LIN {X 0,Y 309.133,Z 1073.835,A -85,B 0,C 180,E1 8987.484,E2 8987.484} C_VEL
LIN {X 0,Y 294.243,Z 1088.868,A -85,B 0,C 180,E1 8985.569,E2 8985.569} C_VEL
LIN {X 0,Y 276.19,Z 1105.751,A -85,B 0,C 180,E1 8982.887,E2 8982.887} C_VEL
LIN {X 0,Y 257.038,Z 1121.964,A -85,B 0,C 180,E1 8979.506,E2 8979.506} C_VEL
LIN {X 0,Y 241.491,Z 1134.247,A -85,B 0,C 180,E1 8976.208,E2 8976.208} C_VEL
LIN {X 0,Y 226.678,Z 1145.297,A -85,B 0,C 180,E1 8972.448,E2 8972.448} C_VEL
LIN {X 0,Y 209.69,Z 1157.432,A -85,B 0,C 180,E1 8967.057,E2 8967.057} C_VEL
LIN {X 0,Y 194.519,Z 1167.62,A -85,B 0,C 180,E1 8960.783,E2 8960.783} C_VEL
LIN {X 0,Y 183.451,Z 1175.062,A -85,B 0,C 180,E1 8954.675,E2 8954.675} C_VEL
LIN {X 0,Y 174.687,Z 1181.102,A -85,B 0,C 180,E1 8948.182,E2 8948.182} C_VEL
LIN {X 0,Y 167.743,Z 1186.26,A -85,B 0,C 180,E1 8940.838,E2 8940.838} C_VEL
LIN {X 0,Y 162.399,Z 1191.034,A -85,B 0,C 180,E1 8931.3,E2 8931.3} C_VEL
LIN {X 0,Y 160.352,Z 1193.692,A -85,B 0,C 180,E1 8922.606,E2 8922.606} C_VEL
LIN {X 0,Y 160.035,Z 1194.885,A -85,B 0,C 180,E1 8915.737,E2 8915.737} C_VEL
LIN {X 0,Y 160.057,Z 1195.249,A -85,B 0,C 180,E1 8909.642,E2 8909.642} C_VEL
LIN {X 0,Y 160.043,Z 1194.803,A -85,B 0,C 180,E1 8903.183,E2 8903.183} C_VEL
LIN {X 0,Y 160.656,Z 1193.192,A -85,B 0,C 180,E1 8895.217,E2 8895.217} C_VEL
LIN {X 0,Y 163.453,Z 1189.886,A -85,B 0,C 180,E1 8886.189,E2 8886.189} C_VEL
LIN {X 0,Y 168.275,Z 1185.792,A -85,B 0,C 180,E1 8878.475,E2 8878.475} C_VEL
LIN {X 0,Y 175.061,Z 1180.789,A -85,B 0,C 180,E1 8871.49,E2 8871.49} C_VEL
LIN {X 0,Y 184.092,Z 1174.573,A -85,B 0,C 180,E1 8864.918,E2 8864.918} C_VEL
LIN {X 0,Y 197.499,Z 1165.629,A -85,B 0,C 180,E1 8857.837,E2 8857.837} C_VEL
LIN {X 0,Y 213.58,Z 1154.53,A -85,B 0,C 180,E1 8851.568,E2 8851.568} C_VEL
LIN {X 0,Y 227.388,Z 1144.675,A -85,B 0,C 180,E1 8847.349,E2 8847.349} C_VEL
LIN {X 0,Y 241.484,Z 1134.135,A -85,B 0,C 180,E1 8843.788,E2 8843.788} C_VEL
LIN {X 0,Y 257.187,Z 1121.707,A -85,B 0,C 180,E1 8840.458,E2 8840.458} C_VEL
LIN {X 0,Y 277.026,Z 1104.8,A -85,B 0,C 180,E1 8836.971,E2 8836.971} C_VEL
LIN {X 0,Y 294.234,Z 1088.677,A -85,B 0,C 180,E1 8834.425,E2 8834.425} C_VEL
LIN {X 0,Y 309.275,Z 1073.464,A -85,B 0,C 180,E1 8832.49,E2 8832.49} C_VEL
LIN {X 0,Y 324.192,Z 1057.141,A -85,B 0,C 180,E1 8830.796,E2 8830.796} C_VEL
LIN {X 0,Y 341.69,Z 1036.137,A -85,B 0,C 180,E1 8829.035,E2 8829.035} C_VEL
LIN {X 0,Y 356.653,Z 1015.961,A -85,B 0,C 180,E1 8827.687,E2 8827.687} C_VEL
LIN {X 0,Y 368.714,Z 998.106,A -85,B 0,C 180,E1 8826.696,E2 8826.696} C_VEL
LIN {X 0,Y 379.924,Z 979.871,A -85,B 0,C 180,E1 8825.85,E2 8825.85} C_VEL
LIN {X 0,Y 390.494,Z 960.848,A -85,B 0,C 180,E1 8825.108,E2 8825.108} C_VEL
LIN {X 0,Y 401.796,Z 938.038,A -85,B 0,C 180,E1 8824.371,E2 8824.371} C_VEL
LIN {X 0,Y 412.803,Z 911.976,A -85,B 0,C 180,E1 8823.706,E2 8823.706} C_VEL
LIN {X 0,Y 420.62,Z 890.255,A -85,B 0,C 180,E1 8823.261,E2 8823.261} C_VEL
LIN {X 0,Y 427.238,Z 868.633,A -85,B 0,C 180,E1 8822.905,E2 8822.905} C_VEL
LIN {X 0,Y 433.159,Z 845.153,A -85,B 0,C 180,E1 8822.584,E2 8822.584} C_VEL
LIN {X 0,Y 438.789,Z 815.012,A -85,B 0,C 180,E1 8822.194,E2 8822.194} C_VEL
LIN {X 0,Y 446.722,Z 751.327,A -85,B 0,C 180,E1 8821.414,E2 8821.414} C_VEL
LIN {X 0,Y 455.842,Z 675.807,A -85,B 0,C 180,E1 8820.471,E2 8820.471} C_VEL
LIN {X 0,Y 455.856,Z 675.472,A -85,B 0,C 180,E1 8819.372,E2 8819.372} C_VEL
LIN {X 0,Y 455.813,Z 675.985,A -85,B 0,C 180,E1 8819.103,E2 8819.103} C_VEL
LIN {X 0,Y 439.212,Z 811.582,A -85,B 0,C 180,E1 8817.459,E2 8817.459} C_VEL
LIN {X 0,Y 434.453,Z 838.722,A -85,B 0,C 180,E1 8817.116,E2 8817.116} C_VEL
LIN {X 0,Y 427.865,Z 865.427,A -85,B 0,C 180,E1 8816.703,E2 8816.703} C_VEL
LIN {X 0,Y 421.567,Z 886.299,A -85,B 0,C 180,E1 8816.301,E2 8816.301} C_VEL
LIN {X 0,Y 414.352,Z 906.676,A -85,B 0,C 180,E1 8815.831,E2 8815.831} C_VEL
LIN {X 0,Y 405.832,Z 927.534,A -85,B 0,C 180,E1 8815.256,E2 8815.256} C_VEL
LIN {X 0,Y 394.302,Z 952.101,A -85,B 0,C 180,E1 8814.434,E2 8814.434} C_VEL
LIN {X 0,Y 381.896,Z 974.697,A -85,B 0,C 180,E1 8813.505,E2 8813.505} C_VEL
LIN {X 0,Y 370.033,Z 994.026,A -85,B 0,C 180,E1 8812.547,E2 8812.547} C_VEL
LIN {X 0,Y 358.475,Z 1011.099,A -85,B 0,C 180,E1 8811.55,E2 8811.55} C_VEL
LIN {X 0,Y 344.895,Z 1029.371,A -85,B 0,C 180,E1 8810.287,E2 8810.287} C_VEL
LIN {X 0,Y 326.629,Z 1051.422,A -85,B 0,C 180,E1 8808.397,E2 8808.397} C_VEL
LIN {X 0,Y 311.406,Z 1067.929,A -85,B 0,C 180,E1 8806.622,E2 8806.622} C_VEL
LIN {X 0,Y 297.374,Z 1081.972,A -85,B 0,C 180,E1 8804.791,E2 8804.791} C_VEL
LIN {X 0,Y 282.808,Z 1095.479,A -85,B 0,C 180,E1 8802.663,E2 8802.663} C_VEL
LIN {X 0,Y 267.028,Z 1109.062,A -85,B 0,C 180,E1 8800.025,E2 8800.025} C_VEL
LIN {X 0,Y 247.214,Z 1124.737,A -85,B 0,C 180,E1 8796.072,E2 8796.072} C_VEL
LIN {X 0,Y 231.552,Z 1136.124,A -85,B 0,C 180,E1 8792.276,E2 8792.276} C_VEL
LIN {X 0,Y 217.635,Z 1145.68,A -85,B 0,C 180,E1 8788.203,E2 8788.203} C_VEL
LIN {X 0,Y 204.25,Z 1154.443,A -85,B 0,C 180,E1 8783.4,E2 8783.4} C_VEL
LIN {X 0,Y 189.786,Z 1163.686,A -85,B 0,C 180,E1 8776.638,E2 8776.638} C_VEL
LIN {X 0,Y 177.958,Z 1170.967,A -85,B 0,C 180,E1 8768.996,E2 8768.996} C_VEL
LIN {X 0,Y 170.605,Z 1175.705,A -85,B 0,C 180,E1 8762.23,E2 8762.23} C_VEL
LIN {X 0,Y 165.299,Z 1179.405,A -85,B 0,C 180,E1 8755.05,E2 8755.05} C_VEL
LIN {X 0,Y 162.12,Z 1181.995,A -85,B 0,C 180,E1 8747.961,E2 8747.961} C_VEL
LIN {X 0,Y 160.603,Z 1183.636,A -85,B 0,C 180,E1 8741.128,E2 8741.128} C_VEL
LIN {X 0,Y 160.127,Z 1184.462,A -85,B 0,C 180,E1 8735.015,E2 8735.015} C_VEL
LIN {X 0,Y 160.068,Z 1184.682,A -85,B 0,C 180,E1 8728.568,E2 8728.568} C_VEL
LIN {X 0,Y 160.302,Z 1184.173,A -85,B 0,C 180,E1 8721.752,E2 8721.752} C_VEL
LIN {X 0,Y 161.666,Z 1182.47,A -85,B 0,C 180,E1 8713.469,E2 8713.469} C_VEL
LIN {X 0,Y 164.853,Z 1179.775,A -85,B 0,C 180,E1 8705.643,E2 8705.643} C_VEL
LIN {X 0,Y 169.941,Z 1176.184,A -85,B 0,C 180,E1 8698.424,E2 8698.424} C_VEL
LIN {X 0,Y 177.089,Z 1171.558,A -85,B 0,C 180,E1 8691.606,E2 8691.606} C_VEL
LIN {X 0,Y 186.7,Z 1165.567,A -85,B 0,C 180,E1 8685.016,E2 8685.016} C_VEL
LIN {X 0,Y 200.602,Z 1156.965,A -85,B 0,C 180,E1 8678.046,E2 8678.046} C_VEL
LIN {X 0,Y 216.185,Z 1146.747,A -85,B 0,C 180,E1 8672.181,E2 8672.181} C_VEL
LIN {X 0,Y 230.378,Z 1137.051,A -85,B 0,C 180,E1 8667.953,E2 8667.953} C_VEL
LIN {X 0,Y 245.568,Z 1126.068,A -85,B 0,C 180,E1 8664.211,E2 8664.211} C_VEL
LIN {X 0,Y 264.596,Z 1111.293,A -85,B 0,C 180,E1 8660.345,E2 8660.345} C_VEL
LIN {X 0,Y 281.866,Z 1096.514,A -85,B 0,C 180,E1 8657.405,E2 8657.405} C_VEL
LIN {X 0,Y 296.484,Z 1083.035,A -85,B 0,C 180,E1 8655.251,E2 8655.251} C_VEL
LIN {X 0,Y 311.317,Z 1068.251,A -85,B 0,C 180,E1 8653.309,E2 8653.309} C_VEL
LIN {X 0,Y 327.453,Z 1050.768,A -85,B 0,C 180,E1 8651.435,E2 8651.435} C_VEL
LIN {X 0,Y 345.095,Z 1029.428,A -85,B 0,C 180,E1 8649.615,E2 8649.615} C_VEL
LIN {X 0,Y 358.749,Z 1011.07,A -85,B 0,C 180,E1 8648.347,E2 8648.347} C_VEL
LIN {X 0,Y 370.481,Z 993.735,A -85,B 0,C 180,E1 8647.338,E2 8647.338} C_VEL
LIN {X 0,Y 382.316,Z 974.425,A -85,B 0,C 180,E1 8646.385,E2 8646.385} C_VEL
LIN {X 0,Y 395.69,Z 949.815,A -85,B 0,C 180,E1 8645.387,E2 8645.387} C_VEL
LIN {X 0,Y 406.271,Z 927.122,A -85,B 0,C 180,E1 8644.638,E2 8644.638} C_VEL
LIN {X 0,Y 414.492,Z 907.01,A -85,B 0,C 180,E1 8644.083,E2 8644.083} C_VEL
LIN {X 0,Y 421.775,Z 886.483,A -85,B 0,C 180,E1 8643.61,E2 8643.61} C_VEL
LIN {X 0,Y 428.306,Z 864.819,A -85,B 0,C 180,E1 8643.194,E2 8643.194} C_VEL
LIN {X 0,Y 434.947,Z 837.545,A -85,B 0,C 180,E1 8642.777,E2 8642.777} C_VEL
LIN {X 0,Y 439.509,Z 811.419,A -85,B 0,C 180,E1 8642.447,E2 8642.447} C_VEL
LIN {X 0,Y 456.081,Z 676.099,A -85,B 0,C 180,E1 8640.786,E2 8640.786} C_VEL
LIN {X 0,Y 456.119,Z 675.624,A -85,B 0,C 180,E1 8640,E2 8640} C_VEL
LIN {X 0,Y 456.064,Z 676.332,A -85,B 0,C 180,E1 8639.494,E2 8639.494} C_VEL
LIN {X 0,Y 447.534,Z 746.879,A -85,B 0,C 180,E1 8638.641,E2 8638.641} C_VEL
LIN {X 0,Y 446.581,Z 754.582,A -85,B 0,C 180,E1 8638.675,E2 8638.675} C_VEL
LIN {X 0,Y 443.952,Z 775.216,A -85,B 0,C 180,E1 8639.235,E2 8639.235} C_VEL
LIN {X 0,Y 443.138,Z 781.824,A -85,B 0,C 180,E1 8639.253,E2 8639.253} C_VEL
LIN {X 0,Y 437.817,Z 821.436,A -85,B 0,C 180,E1 8638.777,E2 8638.777} C_VEL
LIN {X 0,Y 432.44,Z 847.855,A -85,B 0,C 180,E1 8638.445,E2 8638.445} C_VEL
LIN {X 0,Y 426.753,Z 869.852,A -85,B 0,C 180,E1 8638.156,E2 8638.156} C_VEL
LIN {X 0,Y 420.056,Z 891.346,A -85,B 0,C 180,E1 8637.817,E2 8637.817} C_VEL
LIN {X 0,Y 410.398,Z 917.489,A -85,B 0,C 180,E1 8637.295,E2 8637.295} C_VEL
LIN {X 0,Y 399.613,Z 941.699,A -85,B 0,C 180,E1 8636.679,E2 8636.679} C_VEL
LIN {X 0,Y 389.37,Z 961.953,A -85,B 0,C 180,E1 8636.044,E2 8636.044} C_VEL
LIN {X 0,Y 378.147,Z 981.776,A -85,B 0,C 180,E1 8635.298,E2 8635.298} C_VEL
LIN {X 0,Y 364.255,Z 1003.777,A -85,B 0,C 180,E1 8634.289,E2 8634.289} C_VEL
LIN {X 0,Y 347.814,Z 1026.636,A -85,B 0,C 180,E1 8632.978,E2 8632.978} C_VEL
LIN {X 0,Y 333.928,Z 1044.093,A -85,B 0,C 180,E1 8631.736,E2 8631.736} C_VEL
LIN {X 0,Y 320.189,Z 1059.945,A -85,B 0,C 180,E1 8630.383,E2 8630.383} C_VEL
LIN {X 0,Y 304.863,Z 1076.22,A -85,B 0,C 180,E1 8628.704,E2 8628.704} C_VEL
LIN {X 0,Y 285.175,Z 1095.312,A -85,B 0,C 180,E1 8626.206,E2 8626.206} C_VEL
LIN {X 0,Y 267.821,Z 1110.53,A -85,B 0,C 180,E1 8623.629,E2 8623.629} C_VEL
LIN {X 0,Y 251.898,Z 1123.505,A -85,B 0,C 180,E1 8620.855,E2 8620.855} C_VEL
LIN {X 0,Y 235.856,Z 1135.727,A -85,B 0,C 180,E1 8617.542,E2 8617.542} C_VEL
LIN {X 0,Y 217.054,Z 1149.161,A -85,B 0,C 180,E1 8612.754,E2 8612.754} C_VEL
LIN {X 0,Y 200.577,Z 1160.078,A -85,B 0,C 180,E1 8607.399,E2 8607.399} C_VEL
LIN {X 0,Y 187.713,Z 1168.338,A -85,B 0,C 180,E1 8602.029,E2 8602.029} C_VEL
LIN {X 0,Y 176.096,Z 1175.728,A -85,B 0,C 180,E1 8595.677,E2 8595.677} C_VEL
LIN {X 0,Y 164.807,Z 1183.173,A -85,B 0,C 180,E1 8586.914,E2 8586.914} C_VEL
LIN {X 0,Y 157.356,Z 1188.463,A -85,B 0,C 180,E1 8577.636,E2 8577.636} C_VEL
LIN {X 0,Y 153.824,Z 1191.615,A -85,B 0,C 180,E1 8569.755,E2 8569.755} C_VEL
LIN {X 0,Y 152.3,Z 1193.647,A -85,B 0,C 180,E1 8562.127,E2 8562.127} C_VEL
LIN {X 0,Y 152.038,Z 1194.648,A -85,B 0,C 180,E1 8555.661,E2 8555.661} C_VEL
LIN {X 0,Y 152.06,Z 1194.963,A -85,B 0,C 180,E1 8549.246,E2 8549.246} C_VEL
LIN {X 0,Y 152.062,Z 1194.506,A -85,B 0,C 180,E1 8542.443,E2 8542.443} C_VEL
LIN {X 0,Y 152.934,Z 1192.683,A -85,B 0,C 180,E1 8533.673,E2 8533.673} C_VEL
LIN {X 0,Y 155.921,Z 1189.614,A -85,B 0,C 180,E1 8524.961,E2 8524.961} C_VEL
LIN {X 0,Y 161.222,Z 1185.518,A -85,B 0,C 180,E1 8516.924,E2 8516.924} C_VEL
LIN {X 0,Y 168.569,Z 1180.517,A -85,B 0,C 180,E1 8509.72,E2 8509.72} C_VEL
LIN {X 0,Y 178.049,Z 1174.414,A -85,B 0,C 180,E1 8503.111,E2 8503.111} C_VEL
LIN {X 0,Y 191.23,Z 1166.08,A -85,B 0,C 180,E1 8496.371,E2 8496.371} C_VEL
LIN {X 0,Y 208.586,Z 1154.721,A -85,B 0,C 180,E1 8489.817,E2 8489.817} C_VEL
LIN {X 0,Y 223.687,Z 1144.357,A -85,B 0,C 180,E1 8485.412,E2 8485.412} C_VEL
LIN {X 0,Y 238.203,Z 1133.856,A -85,B 0,C 180,E1 8481.929,E2 8481.929} C_VEL
LIN {X 0,Y 254.364,Z 1121.429,A -85,B 0,C 180,E1 8478.68,E2 8478.68} C_VEL
LIN {X 0,Y 274.693,Z 1104.522,A -85,B 0,C 180,E1 8475.297,E2 8475.297} C_VEL
LIN {X 0,Y 292.263,Z 1088.4,A -85,B 0,C 180,E1 8472.836,E2 8472.836} C_VEL
LIN {X 0,Y 307.578,Z 1073.188,A -85,B 0,C 180,E1 8470.972,E2 8470.972} C_VEL
LIN {X 0,Y 322.534,Z 1057.09,A -85,B 0,C 180,E1 8469.365,E2 8469.365} C_VEL
LIN {X 0,Y 340.019,Z 1036.476,A -85,B 0,C 180,E1 8467.702,E2 8467.702} C_VEL
LIN {X 0,Y 355.458,Z 1015.952,A -85,B 0,C 180,E1 8466.387,E2 8466.387} C_VEL
LIN {X 0,Y 368.085,Z 997.464,A -85,B 0,C 180,E1 8465.409,E2 8465.409} C_VEL
LIN {X 0,Y 379.661,Z 978.78,A -85,B 0,C 180,E1 8464.587,E2 8464.587} C_VEL
LIN {X 0,Y 391.362,Z 957.767,A -85,B 0,C 180,E1 8463.819,E2 8463.819} C_VEL
LIN {X 0,Y 404.015,Z 931.651,A -85,B 0,C 180,E1 8463.053,E2 8463.053} C_VEL
LIN {X 0,Y 413.342,Z 909.121,A -85,B 0,C 180,E1 8462.528,E2 8462.528} C_VEL
LIN {X 0,Y 420.591,Z 888.917,A -85,B 0,C 180,E1 8462.143,E2 8462.143} C_VEL
LIN {X 0,Y 427.152,Z 867.489,A -85,B 0,C 180,E1 8461.813,E2 8461.813} C_VEL
LIN {X 0,Y 433.674,Z 841.477,A -85,B 0,C 180,E1 8461.475,E2 8461.475} C_VEL
LIN {X 0,Y 438.74,Z 813.437,A -85,B 0,C 180,E1 8461.126,E2 8461.126} C_VEL
LIN {X 0,Y 449.767,Z 725.044,A -85,B 0,C 180,E1 8460.073,E2 8460.073} C_VEL
LIN {X 0,Y 452.539,Z 702.413,A -85,B 0,C 180,E1 8459.801,E2 8459.801} C_VEL
LIN {X 0,Y 438.884,Z 812.187,A -85,B 0,C 180,E1 8458.499,E2 8458.499} C_VEL
LIN {X 0,Y 433.988,Z 839.631,A -85,B 0,C 180,E1 8458.163,E2 8458.163} C_VEL
LIN {X 0,Y 427.417,Z 865.917,A -85,B 0,C 180,E1 8457.773,E2 8457.773} C_VEL
LIN {X 0,Y 421.125,Z 886.572,A -85,B 0,C 180,E1 8457.392,E2 8457.392} C_VEL
LIN {X 0,Y 413.79,Z 907.091,A -85,B 0,C 180,E1 8456.939,E2 8456.939} C_VEL
LIN {X 0,Y 405.245,Z 927.806,A -85,B 0,C 180,E1 8456.392,E2 8456.392} C_VEL
LIN {X 0,Y 393.601,Z 952.371,A -85,B 0,C 180,E1 8455.605,E2 8455.605} C_VEL
LIN {X 0,Y 380.583,Z 975.773,A -85,B 0,C 180,E1 8454.682,E2 8454.682} C_VEL
LIN {X 0,Y 369.104,Z 994.24,A -85,B 0,C 180,E1 8453.802,E2 8453.802} C_VEL
LIN {X 0,Y 357.239,Z 1011.55,A -85,B 0,C 180,E1 8452.834,E2 8452.834} C_VEL
LIN {X 0,Y 343.142,Z 1030.245,A -85,B 0,C 180,E1 8451.588,E2 8451.588} C_VEL
LIN {X 0,Y 324.158,Z 1052.696,A -85,B 0,C 180,E1 8449.719,E2 8449.719} C_VEL
LIN {X 0,Y 309.168,Z 1068.643,A -85,B 0,C 180,E1 8448.054,E2 8448.054} C_VEL
LIN {X 0,Y 294.43,Z 1083.078,A -85,B 0,C 180,E1 8446.223,E2 8446.223} C_VEL
LIN {X 0,Y 278.729,Z 1097.27,A -85,B 0,C 180,E1 8444.022,E2 8444.022} C_VEL
LIN {X 0,Y 259.332,Z 1113.38,A -85,B 0,C 180,E1 8440.839,E2 8440.839} C_VEL
LIN {X 0,Y 241.587,Z 1126.697,A -85,B 0,C 180,E1 8437.358,E2 8437.358} C_VEL
LIN {X 0,Y 226.303,Z 1137.406,A -85,B 0,C 180,E1 8433.753,E2 8433.753} C_VEL
LIN {X 0,Y 211.971,Z 1146.85,A -85,B 0,C 180,E1 8429.678,E2 8429.678} C_VEL
LIN {X 0,Y 195.666,Z 1157.081,A -85,B 0,C 180,E1 8423.841,E2 8423.841} C_VEL
LIN {X 0,Y 180.793,Z 1165.837,A -85,B 0,C 180,E1 8416.702,E2 8416.702} C_VEL
LIN {X 0,Y 170.741,Z 1171.729,A -85,B 0,C 180,E1 8410.103,E2 8410.103} C_VEL
LIN {X 0,Y 163.029,Z 1176.372,A -85,B 0,C 180,E1 8403.082,E2 8403.082} C_VEL
LIN {X 0,Y 157.245,Z 1180.13,A -85,B 0,C 180,E1 8395.216,E2 8395.216} C_VEL
LIN {X 0,Y 153.683,Z 1182.906,A -85,B 0,C 180,E1 8386.634,E2 8386.634} C_VEL
LIN {X 0,Y 152.289,Z 1184.538,A -85,B 0,C 180,E1 8377.925,E2 8377.925} C_VEL
LIN {X 0,Y 152.068,Z 1184.979,A -85,B 0,C 180,E1 8370.753,E2 8370.753} C_VEL
LIN {X 0,Y 152.168,Z 1184.695,A -85,B 0,C 180,E1 8363.965,E2 8363.965} C_VEL
LIN {X 0,Y 153.046,Z 1183.553,A -85,B 0,C 180,E1 8356.012,E2 8356.012} C_VEL
LIN {X 0,Y 156.409,Z 1180.803,A -85,B 0,C 180,E1 8346.251,E2 8346.251} C_VEL
LIN {X 0,Y 162.424,Z 1176.793,A -85,B 0,C 180,E1 8337.499,E2 8337.499} C_VEL
LIN {X 0,Y 170.245,Z 1172.074,A -85,B 0,C 180,E1 8330.196,E2 8330.196} C_VEL
LIN {X 0,Y 179.885,Z 1166.425,A -85,B 0,C 180,E1 8323.732,E2 8323.732} C_VEL
LIN {X 0,Y 192.557,Z 1158.974,A -85,B 0,C 180,E1 8317.396,E2 8317.396} C_VEL
LIN {X 0,Y 210.484,Z 1147.915,A -85,B 0,C 180,E1 8310.706,E2 8310.706} C_VEL
LIN {X 0,Y 225.875,Z 1137.807,A -85,B 0,C 180,E1 8306.275,E2 8306.275} C_VEL
LIN {X 0,Y 240.913,Z 1127.307,A -85,B 0,C 180,E1 8302.705,E2 8302.705} C_VEL
LIN {X 0,Y 257.581,Z 1114.852,A -85,B 0,C 180,E1 8299.395,E2 8299.395} C_VEL
LIN {X 0,Y 277.778,Z 1098.3,A -85,B 0,C 180,E1 8296.042,E2 8296.042} C_VEL
LIN {X 0,Y 293.784,Z 1083.901,A -85,B 0,C 180,E1 8293.783,E2 8293.783} C_VEL
LIN {X 0,Y 308.622,Z 1069.432,A -85,B 0,C 180,E1 8291.93,E2 8291.93} C_VEL
LIN {X 0,Y 323.765,Z 1053.386,A -85,B 0,C 180,E1 8290.243,E2 8290.243} C_VEL
LIN {X 0,Y 341.679,Z 1032.458,A -85,B 0,C 180,E1 8288.472,E2 8288.472} C_VEL
LIN {X 0,Y 356.71,Z 1012.656,A -85,B 0,C 180,E1 8287.135,E2 8287.135} C_VEL
LIN {X 0,Y 368.576,Z 995.454,A -85,B 0,C 180,E1 8286.162,E2 8286.162} C_VEL
LIN {X 0,Y 380.009,Z 977.185,A -85,B 0,C 180,E1 8285.284,E2 8285.284} C_VEL
LIN {X 0,Y 390.773,Z 958.083,A -85,B 0,C 180,E1 8284.508,E2 8284.508} C_VEL
LIN {X 0,Y 402.781,Z 934.091,A -85,B 0,C 180,E1 8283.699,E2 8283.699} C_VEL
LIN {X 0,Y 413.183,Z 909.393,A -85,B 0,C 180,E1 8283.024,E2 8283.024} C_VEL
LIN {X 0,Y 420.855,Z 888.21,A -85,B 0,C 180,E1 8282.549,E2 8282.549} C_VEL
LIN {X 0,Y 427.316,Z 867.242,A -85,B 0,C 180,E1 8282.158,E2 8282.158} C_VEL
LIN {X 0,Y 433.051,Z 844.755,A -85,B 0,C 180,E1 8281.815,E2 8281.815} C_VEL
LIN {X 0,Y 438.774,Z 814.893,A -85,B 0,C 180,E1 8281.442,E2 8281.442} C_VEL
LIN {X 0,Y 445.925,Z 758.797,A -85,B 0,C 180,E1 8280.774,E2 8280.774} C_VEL
LIN {X 0,Y 452.345,Z 706.338,A -85,B 0,C 180,E1 8280.15,E2 8280.15} C_VEL
LIN {X 0,Y 443.138,Z 781.824,A -85,B 0,C 180,E1 8279.253,E2 8279.253} C_VEL
LIN {X 0,Y 442.206,Z 789.524,A -85,B 0,C 180,E1 8279.294,E2 8279.294} C_VEL
LIN {X 0,Y 439.396,Z 810.123,A -85,B 0,C 180,E1 8279.867,E2 8279.867} C_VEL
LIN {X 0,Y 438.423,Z 816.713,A -85,B 0,C 180,E1 8279.884,E2 8279.884} C_VEL
LIN {X 0,Y 432.733,Z 845.774,A -85,B 0,C 180,E1 8279.534,E2 8279.534} C_VEL
LIN {X 0,Y 426.874,Z 868.532,A -85,B 0,C 180,E1 8279.252,E2 8279.252} C_VEL
LIN {X 0,Y 420.383,Z 889.422,A -85,B 0,C 180,E1 8278.946,E2 8278.946} C_VEL
LIN {X 0,Y 412.571,Z 910.848,A -85,B 0,C 180,E1 8278.556,E2 8278.556} C_VEL
LIN {X 0,Y 401.198,Z 937.398,A -85,B 0,C 180,E1 8277.951,E2 8277.951} C_VEL
LIN {X 0,Y 389.875,Z 959.878,A -85,B 0,C 180,E1 8277.302,E2 8277.302} C_VEL
LIN {X 0,Y 379.099,Z 978.945,A -85,B 0,C 180,E1 8276.634,E2 8276.634} C_VEL
LIN {X 0,Y 367.388,Z 997.617,A -85,B 0,C 180,E1 8275.854,E2 8275.854} C_VEL
LIN {X 0,Y 353.868,Z 1017.113,A -85,B 0,C 180,E1 8274.866,E2 8274.866} C_VEL
LIN {X 0,Y 336.157,Z 1039.909,A -85,B 0,C 180,E1 8273.432,E2 8273.432} C_VEL
LIN {X 0,Y 320.61,Z 1057.808,A -85,B 0,C 180,E1 8272.024,E2 8272.024} C_VEL
LIN {X 0,Y 305.578,Z 1073.672,A -85,B 0,C 180,E1 8270.496,E2 8270.496} C_VEL
LIN {X 0,Y 289.583,Z 1089.215,A -85,B 0,C 180,E1 8268.649,E2 8268.649} C_VEL
LIN {X 0,Y 269.96,Z 1106.694,A -85,B 0,C 180,E1 8266.018,E2 8266.018} C_VEL
LIN {X 0,Y 250.952,Z 1121.936,A -85,B 0,C 180,E1 8262.983,E2 8262.983} C_VEL
LIN {X 0,Y 235.188,Z 1133.696,A -85,B 0,C 180,E1 8259.974,E2 8259.974} C_VEL
LIN {X 0,Y 219.288,Z 1144.804,A -85,B 0,C 180,E1 8256.343,E2 8256.343} C_VEL
LIN {X 0,Y 200.986,Z 1156.879,A -85,B 0,C 180,E1 8251.111,E2 8251.111} C_VEL
LIN {X 0,Y 184.478,Z 1166.968,A -85,B 0,C 180,E1 8244.926,E2 8244.926} C_VEL
LIN {X 0,Y 171.871,Z 1174.51,A -85,B 0,C 180,E1 8238.63,E2 8238.63} C_VEL
LIN {X 0,Y 161.828,Z 1180.552,A -85,B 0,C 180,E1 8231.857,E2 8231.857} C_VEL
LIN {X 0,Y 153.35,Z 1185.93,A -85,B 0,C 180,E1 8223.656,E2 8223.656} C_VEL
LIN {X 0,Y 146.994,Z 1190.615,A -85,B 0,C 180,E1 8213.236,E2 8213.236} C_VEL
LIN {X 0,Y 144.513,Z 1193.158,A -85,B 0,C 180,E1 8204.014,E2 8204.014} C_VEL
LIN {X 0,Y 144.045,Z 1194.358,A -85,B 0,C 180,E1 8196.376,E2 8196.376} C_VEL
LIN {X 0,Y 144.065,Z 1194.724,A -85,B 0,C 180,E1 8189.602,E2 8189.602} C_VEL
LIN {X 0,Y 144.055,Z 1194.301,A -85,B 0,C 180,E1 8182.823,E2 8182.823} C_VEL
LIN {X 0,Y 144.847,Z 1192.768,A -85,B 0,C 180,E1 8173.972,E2 8173.972} C_VEL
LIN {X 0,Y 148.469,Z 1189.342,A -85,B 0,C 180,E1 8163.61,E2 8163.61} C_VEL
LIN {X 0,Y 154.293,Z 1185.243,A -85,B 0,C 180,E1 8155.232,E2 8155.232} C_VEL
LIN {X 0,Y 162.554,Z 1180.06,A -85,B 0,C 180,E1 8147.573,E2 8147.573} C_VEL
LIN {X 0,Y 172.925,Z 1173.822,A -85,B 0,C 180,E1 8140.761,E2 8140.761} C_VEL
LIN {X 0,Y 188.241,Z 1164.705,A -85,B 0,C 180,E1 8133.497,E2 8133.497} C_VEL
LIN {X 0,Y 205.231,Z 1153.972,A -85,B 0,C 180,E1 8127.541,E2 8127.541} C_VEL
LIN {X 0,Y 220.138,Z 1144.117,A -85,B 0,C 180,E1 8123.441,E2 8123.441} C_VEL
LIN {X 0,Y 235.181,Z 1133.578,A -85,B 0,C 180,E1 8120.021,E2 8120.021} C_VEL
LIN {X 0,Y 251.92,Z 1121.054,A -85,B 0,C 180,E1 8116.843,E2 8116.843} C_VEL
LIN {X 0,Y 272.81,Z 1104.059,A -85,B 0,C 180,E1 8113.566,E2 8113.566} C_VEL
LIN {X 0,Y 290.52,Z 1088.123,A -85,B 0,C 180,E1 8111.229,E2 8111.229} C_VEL
LIN {X 0,Y 306.101,Z 1072.911,A -85,B 0,C 180,E1 8109.44,E2 8109.44} C_VEL
LIN {X 0,Y 321.72,Z 1056.338,A -85,B 0,C 180,E1 8107.86,E2 8107.86} C_VEL
LIN {X 0,Y 339.96,Z 1034.971,A -85,B 0,C 180,E1 8106.232,E2 8106.232} C_VEL
LIN {X 0,Y 354.826,Z 1015.412,A -85,B 0,C 180,E1 8105.051,E2 8105.051} C_VEL
LIN {X 0,Y 367.208,Z 997.487,A -85,B 0,C 180,E1 8104.148,E2 8104.148} C_VEL
LIN {X 0,Y 378.606,Z 979.324,A -85,B 0,C 180,E1 8103.386,E2 8103.386} C_VEL
LIN {X 0,Y 389.381,Z 960.301,A -85,B 0,C 180,E1 8102.717,E2 8102.717} C_VEL
LIN {X 0,Y 400.702,Z 937.866,A -85,B 0,C 180,E1 8102.065,E2 8102.065} C_VEL
LIN {X 0,Y 412.074,Z 911.428,A -85,B 0,C 180,E1 8101.458,E2 8101.458} C_VEL
LIN {X 0,Y 420.011,Z 889.706,A -85,B 0,C 180,E1 8101.06,E2 8101.06} C_VEL
LIN {X 0,Y 426.689,Z 868.206,A -85,B 0,C 180,E1 8100.746,E2 8100.746} C_VEL
LIN {X 0,Y 432.67,Z 844.86,A -85,B 0,C 180,E1 8100.456,E2 8100.456} C_VEL
LIN {X 0,Y 438.452,Z 814.548,A -85,B 0,C 180,E1 8100.091,E2 8100.091} C_VEL
LIN {X 0,Y 441.751,Z 790.273,A -85,B 0,C 180,E1 8099.803,E2 8099.803} C_VEL
LIN {X 0,Y 436.617,Z 825.351,A -85,B 0,C 180,E1 8099.394,E2 8099.394} C_VEL
LIN {X 0,Y 431.802,Z 848.29,A -85,B 0,C 180,E1 8099.11,E2 8099.11} C_VEL
LIN {X 0,Y 426.226,Z 869.517,A -85,B 0,C 180,E1 8098.794,E2 8098.794} C_VEL
LIN {X 0,Y 419.353,Z 891.263,A -85,B 0,C 180,E1 8098.398,E2 8098.398} C_VEL
LIN {X 0,Y 409.243,Z 917.962,A -85,B 0,C 180,E1 8097.797,E2 8097.797} C_VEL
LIN {X 0,Y 398.973,Z 940.651,A -85,B 0,C 180,E1 8097.164,E2 8097.164} C_VEL
LIN {X 0,Y 389.157,Z 959.792,A -85,B 0,C 180,E1 8096.529,E2 8096.529} C_VEL
LIN {X 0,Y 378.533,Z 978.342,A -85,B 0,C 180,E1 8095.803,E2 8095.803} C_VEL
LIN {X 0,Y 366.389,Z 997.425,A -85,B 0,C 180,E1 8094.915,E2 8094.915} C_VEL
LIN {X 0,Y 350.704,Z 1019.538,A -85,B 0,C 180,E1 8093.669,E2 8093.669} C_VEL
LIN {X 0,Y 334.555,Z 1039.558,A -85,B 0,C 180,E1 8092.271,E2 8092.271} C_VEL
LIN {X 0,Y 320.003,Z 1055.973,A -85,B 0,C 180,E1 8090.876,E2 8090.876} C_VEL
LIN {X 0,Y 305.265,Z 1071.216,A -85,B 0,C 180,E1 8089.299,E2 8089.299} C_VEL
LIN {X 0,Y 288.089,Z 1087.516,A -85,B 0,C 180,E1 8087.226,E2 8087.226} C_VEL
LIN {X 0,Y 267.84,Z 1104.792,A -85,B 0,C 180,E1 8084.391,E2 8084.391} C_VEL
LIN {X 0,Y 251.56,Z 1117.475,A -85,B 0,C 180,E1 8081.699,E2 8081.699} C_VEL
LIN {X 0,Y 236.087,Z 1128.657,A -85,B 0,C 180,E1 8078.705,E2 8078.705} C_VEL
LIN {X 0,Y 220.01,Z 1139.482,A -85,B 0,C 180,E1 8074.997,E2 8074.997} C_VEL
LIN {X 0,Y 200.845,Z 1151.45,A -85,B 0,C 180,E1 8069.456,E2 8069.456} C_VEL
LIN {X 0,Y 185.401,Z 1160.387,A -85,B 0,C 180,E1 8063.612,E2 8063.612} C_VEL
LIN {X 0,Y 173.261,Z 1167.165,A -85,B 0,C 180,E1 8057.618,E2 8057.618} C_VEL
LIN {X 0,Y 162.727,Z 1172.981,A -85,B 0,C 180,E1 8050.64,E2 8050.64} C_VEL
LIN {X 0,Y 152.993,Z 1178.584,A -85,B 0,C 180,E1 8041.084,E2 8041.084} C_VEL
LIN {X 0,Y 147.146,Z 1182.211,A -85,B 0,C 180,E1 8031.108,E2 8031.108} C_VEL
LIN {X 0,Y 144.901,Z 1184.041,A -85,B 0,C 180,E1 8023.162,E2 8023.162} C_VEL
LIN {X 0,Y 144.155,Z 1184.989,A -85,B 0,C 180,E1 8015.572,E2 8015.572} C_VEL
LIN {X 0,Y 144.073,Z 1185.229,A -85,B 0,C 180,E1 8008.807,E2 8008.807} C_VEL
LIN {X 0,Y 144.346,Z 1184.766,A -85,B 0,C 180,E1 8001.235,E2 8001.235} C_VEL
LIN {X 0,Y 146.007,Z 1183.112,A -85,B 0,C 180,E1 7992.052,E2 7992.052} C_VEL
LIN {X 0,Y 149.822,Z 1180.457,A -85,B 0,C 180,E1 7983.419,E2 7983.419} C_VEL
LIN {X 0,Y 156.106,Z 1176.725,A -85,B 0,C 180,E1 7975.247,E2 7975.247} C_VEL
LIN {X 0,Y 164.704,Z 1171.935,A -85,B 0,C 180,E1 7967.786,E2 7967.786} C_VEL
LIN {X 0,Y 176.413,Z 1165.527,A -85,B 0,C 180,E1 7960.583,E2 7960.583} C_VEL
LIN {X 0,Y 193.349,Z 1155.934,A -85,B 0,C 180,E1 7953.097,E2 7953.097} C_VEL
LIN {X 0,Y 208.499,Z 1146.844,A -85,B 0,C 180,E1 7948.071,E2 7948.071} C_VEL
LIN {X 0,Y 223.729,Z 1137.148,A -85,B 0,C 180,E1 7943.998,E2 7943.998} C_VEL
LIN {X 0,Y 240.84,Z 1125.488,A -85,B 0,C 180,E1 7940.241,E2 7940.241} C_VEL
LIN {X 0,Y 261.726,Z 1109.857,A -85,B 0,C 180,E1 7936.488,E2 7936.488} C_VEL
LIN {X 0,Y 278.234,Z 1096.295,A -85,B 0,C 180,E1 7934.007,E2 7934.007} C_VEL
LIN {X 0,Y 293.702,Z 1082.524,A -85,B 0,C 180,E1 7931.986,E2 7931.986} C_VEL
LIN {X 0,Y 309.781,Z 1066.958,A -85,B 0,C 180,E1 7930.126,E2 7930.126} C_VEL
LIN {X 0,Y 329.275,Z 1046.031,A -85,B 0,C 180,E1 7928.146,E2 7928.146} C_VEL
LIN {X 0,Y 344.356,Z 1027.907,A -85,B 0,C 180,E1 7926.777,E2 7926.777} C_VEL
LIN {X 0,Y 357.701,Z 1010.274,A -85,B 0,C 180,E1 7925.675,E2 7925.675} C_VEL
LIN {X 0,Y 370.205,Z 992.073,A -85,B 0,C 180,E1 7924.727,E2 7924.727} C_VEL
LIN {X 0,Y 384.249,Z 969.301,A -85,B 0,C 180,E1 7923.73,E2 7923.73} C_VEL
LIN {X 0,Y 396.923,Z 945.387,A -85,B 0,C 180,E1 7922.888,E2 7922.888} C_VEL
LIN {X 0,Y 406.269,Z 925.389,A -85,B 0,C 180,E1 7922.304,E2 7922.304} C_VEL
LIN {X 0,Y 414.758,Z 904.672,A -85,B 0,C 180,E1 7921.796,E2 7921.796} C_VEL
LIN {X 0,Y 423.05,Z 881.097,A -85,B 0,C 180,E1 7921.315,E2 7921.315} C_VEL
LIN {X 0,Y 430.893,Z 853.28,A -85,B 0,C 180,E1 7920.866,E2 7920.866} C_VEL
LIN {X 0,Y 435.896,Z 830.591,A -85,B 0,C 180,E1 7920.578,E2 7920.578} C_VEL
LIN {X 0,Y 439.63,Z 808.378,A -85,B 0,C 180,E1 7920.317,E2 7920.317} C_VEL
LIN {X 0,Y 441.563,Z 794.154,A -85,B 0,C 180,E1 7920.148,E2 7920.148} C_VEL
LIN {X 0,Y 438.423,Z 816.713,A -85,B 0,C 180,E1 7919.884,E2 7919.884} C_VEL
LIN {X 0,Y 438.399,Z 817.05,A -85,B 0,C 180,E1 7919.882,E2 7919.882} C_VEL
LIN {X 0,Y 438.399,Z 899.547,A -85,B 0,C 180,E1 7919.882,E2 7919.882} C_VEL
LIN {X 0,Y 429.245,Z 899.547,A -85,B 0,C 180,E1 7920.272,E2 7920.272} C_VEL
LIN {X 0,Y 427.344,Z 897.547,A -85,B 0,C 180,E1 7920.356,E2 7920.356} C_VEL
LIN {X 0,Y 427.344,Z 879.903,A -85,B 0,C 180,E1 7920.356,E2 7920.356} C_VEL
LIN {X 0,Y 423.659,Z 879.234,A -85,B 0,C 180,E1 7920.19,E2 7920.19} C_VEL
LIN {X 0,Y 414.942,Z 904.142,A -85,B 0,C 180,E1 7919.8,E2 7919.8} C_VEL
LIN {X 0,Y 406.464,Z 924.919,A -85,B 0,C 180,E1 7919.39,E2 7919.39} C_VEL
LIN {X 0,Y 397.511,Z 944.209,A -85,B 0,C 180,E1 7918.932,E2 7918.932} C_VEL
LIN {X 0,Y 387.102,Z 964.146,A -85,B 0,C 180,E1 7918.359,E2 7918.359} C_VEL
LIN {X 0,Y 373.291,Z 987.669,A -85,B 0,C 180,E1 7917.535,E2 7917.535} C_VEL
LIN {X 0,Y 358.302,Z 1009.835,A -85,B 0,C 180,E1 7916.553,E2 7916.553} C_VEL
LIN {X 0,Y 344.482,Z 1028.259,A -85,B 0,C 180,E1 7915.563,E2 7915.563} C_VEL
LIN {X 0,Y 330.487,Z 1045.269,A -85,B 0,C 180,E1 7914.444,E2 7914.444} C_VEL
LIN {X 0,Y 314.951,Z 1062.521,A -85,B 0,C 180,E1 7913.071,E2 7913.071} C_VEL
LIN {X 0,Y 294.577,Z 1082.91,A -85,B 0,C 180,E1 7911.009,E2 7911.009} C_VEL
LIN {X 0,Y 277.324,Z 1098.474,A -85,B 0,C 180,E1 7908.983,E2 7908.983} C_VEL
LIN {X 0,Y 261.794,Z 1111.407,A -85,B 0,C 180,E1 7906.882,E2 7906.882} C_VEL
LIN {X 0,Y 245.158,Z 1124.249,A -85,B 0,C 180,E1 7904.26,E2 7904.26} C_VEL
LIN {X 0,Y 224.997,Z 1138.674,A -85,B 0,C 180,E1 7900.407,E2 7900.407} C_VEL
LIN {X 0,Y 206,Z 1150.963,A -85,B 0,C 180,E1 7895.851,E2 7895.851} C_VEL
LIN {X 0,Y 190.586,Z 1160.359,A -85,B 0,C 180,E1 7891.177,E2 7891.177} C_VEL
LIN {X 0,Y 176.553,Z 1168.515,A -85,B 0,C 180,E1 7885.774,E2 7885.774} C_VEL
LIN {X 0,Y 161.906,Z 1176.857,A -85,B 0,C 180,E1 7878.165,E2 7878.165} C_VEL
LIN {X 0,Y 149.745,Z 1183.708,A -85,B 0,C 180,E1 7868.876,E2 7868.876} C_VEL
LIN {X 0,Y 142.585,Z 1188.088,A -85,B 0,C 180,E1 7860.324,E2 7860.324} C_VEL
LIN {X 0,Y 138.301,Z 1191.197,A -85,B 0,C 180,E1 7851.636,E2 7851.636} C_VEL
LIN {X 0,Y 136.443,Z 1193.114,A -85,B 0,C 180,E1 7843.562,E2 7843.562} C_VEL
LIN {X 0,Y 136.048,Z 1194.12,A -85,B 0,C 180,E1 7836.329,E2 7836.329} C_VEL
LIN {X 0,Y 136.069,Z 1194.461,A -85,B 0,C 180,E1 7829.579,E2 7829.579} C_VEL
LIN {X 0,Y 136.07,Z 1194.036,A -85,B 0,C 180,E1 7822.399,E2 7822.399} C_VEL
LIN {X 0,Y 137.044,Z 1192.469,A -85,B 0,C 180,E1 7812.902,E2 7812.902} C_VEL
LIN {X 0,Y 141.103,Z 1189.07,A -85,B 0,C 180,E1 7802.117,E2 7802.117} C_VEL
LIN {X 0,Y 147.513,Z 1184.968,A -85,B 0,C 180,E1 7793.382,E2 7793.382} C_VEL
LIN {X 0,Y 156.138,Z 1179.964,A -85,B 0,C 180,E1 7785.733,E2 7785.733} C_VEL
LIN {X 0,Y 166.975,Z 1173.859,A -85,B 0,C 180,E1 7778.881,E2 7778.881} C_VEL
LIN {X 0,Y 181.059,Z 1165.888,A -85,B 0,C 180,E1 7772.338,E2 7772.338} C_VEL
LIN {X 0,Y 200.716,Z 1154.163,A -85,B 0,C 180,E1 7765.626,E2 7765.626} C_VEL
LIN {X 0,Y 216.918,Z 1143.838,A -85,B 0,C 180,E1 7761.395,E2 7761.395} C_VEL
LIN {X 0,Y 232.634,Z 1133.155,A -85,B 0,C 180,E1 7758.027,E2 7758.027} C_VEL
LIN {X 0,Y 249.482,Z 1120.872,A -85,B 0,C 180,E1 7755.015,E2 7755.015} C_VEL
LIN {X 0,Y 270.751,Z 1103.966,A -85,B 0,C 180,E1 7751.87,E2 7751.87} C_VEL
LIN {X 0,Y 289.009,Z 1087.846,A -85,B 0,C 180,E1 7749.603,E2 7749.603} C_VEL
LIN {X 0,Y 304.526,Z 1072.953,A -85,B 0,C 180,E1 7747.927,E2 7747.927} C_VEL
LIN {X 0,Y 319.981,Z 1056.826,A -85,B 0,C 180,E1 7746.452,E2 7746.452} C_VEL
LIN {X 0,Y 337.716,Z 1036.532,A -85,B 0,C 180,E1 7744.96,E2 7744.96} C_VEL
LIN {X 0,Y 354.221,Z 1015.105,A -85,B 0,C 180,E1 7743.723,E2 7743.723} C_VEL
LIN {X 0,Y 366.903,Z 996.917,A -85,B 0,C 180,E1 7742.856,E2 7742.856} C_VEL
LIN {X 0,Y 378.726,Z 978.196,A -85,B 0,C 180,E1 7742.118,E2 7742.118} C_VEL
LIN {X 0,Y 390.566,Z 957.311,A -85,B 0,C 180,E1 7741.435,E2 7741.435} C_VEL
LIN {X 0,Y 403.476,Z 931.104,A -85,B 0,C 180,E1 7740.751,E2 7740.751} C_VEL
LIN {X 0,Y 412.945,Z 908.574,A -85,B 0,C 180,E1 7740.283,E2 7740.283} C_VEL
LIN {X 0,Y 420.587,Z 887.509,A -85,B 0,C 180,E1 7739.929,E2 7739.929} C_VEL
LIN {X 0,Y 424.192,Z 876.509,A -85,B 0,C 180,E1 7739.765,E2 7739.765} C_VEL
LIN {X 0,Y 414.974,Z 903.186,A -85,B 0,C 180,E1 7739.261,E2 7739.261} C_VEL
LIN {X 0,Y 406.532,Z 923.853,A -85,B 0,C 180,E1 7738.785,E2 7738.785} C_VEL
LIN {X 0,Y 397.131,Z 944.002,A -85,B 0,C 180,E1 7738.232,E2 7738.232} C_VEL
LIN {X 0,Y 386.293,Z 964.531,A -85,B 0,C 180,E1 7737.564,E2 7737.564} C_VEL
LIN {X 0,Y 371.605,Z 988.956,A -85,B 0,C 180,E1 7736.588,E2 7736.588} C_VEL
LIN {X 0,Y 357.507,Z 1009.448,A -85,B 0,C 180,E1 7735.589,E2 7735.589} C_VEL
LIN {X 0,Y 344.011,Z 1027.177,A -85,B 0,C 180,E1 7734.54,E2 7734.54} C_VEL
LIN {X 0,Y 330.162,Z 1043.742,A -85,B 0,C 180,E1 7733.367,E2 7733.367} C_VEL
LIN {X 0,Y 312.24,Z 1063.249,A -85,B 0,C 180,E1 7731.682,E2 7731.682} C_VEL
LIN {X 0,Y 293.686,Z 1081.128,A -85,B 0,C 180,E1 7729.705,E2 7729.705} C_VEL
LIN {X 0,Y 277.318,Z 1095.544,A -85,B 0,C 180,E1 7727.708,E2 7727.708} C_VEL
LIN {X 0,Y 261.322,Z 1108.51,A -85,B 0,C 180,E1 7725.469,E2 7725.469} C_VEL
LIN {X 0,Y 242.377,Z 1122.655,A -85,B 0,C 180,E1 7722.349,E2 7722.349} C_VEL
LIN {X 0,Y 221.818,Z 1136.448,A -85,B 0,C 180,E1 7718.211,E2 7718.211} C_VEL
LIN {X 0,Y 206.292,Z 1146.06,A -85,B 0,C 180,E1 7714.356,E2 7714.356} C_VEL
LIN {X 0,Y 191.789,Z 1154.48,A -85,B 0,C 180,E1 7709.929,E2 7709.929} C_VEL
LIN {X 0,Y 177.862,Z 1162.125,A -85,B 0,C 180,E1 7704.599,E2 7704.599} C_VEL
LIN {X 0,Y 162.911,Z 1170.069,A -85,B 0,C 180,E1 7696.916,E2 7696.916} C_VEL
LIN {X 0,Y 150.934,Z 1176.151,A -85,B 0,C 180,E1 7687.969,E2 7687.969} C_VEL
LIN {X 0,Y 143.61,Z 1180.065,A -85,B 0,C 180,E1 7679.625,E2 7679.625} C_VEL
LIN {X 0,Y 139.043,Z 1182.799,A -85,B 0,C 180,E1 7671.072,E2 7671.072} C_VEL
LIN {X 0,Y 136.876,Z 1184.433,A -85,B 0,C 180,E1 7663.088,E2 7663.088} C_VEL
LIN {X 0,Y 136.173,Z 1185.252,A -85,B 0,C 180,E1 7655.9,E2 7655.9} C_VEL
LIN {X 0,Y 136.078,Z 1185.491,A -85,B 0,C 180,E1 7648.737,E2 7648.737} C_VEL
LIN {X 0,Y 136.39,Z 1185.03,A -85,B 0,C 180,E1 7640.719,E2 7640.719} C_VEL
LIN {X 0,Y 138.28,Z 1183.379,A -85,B 0,C 180,E1 7631.012,E2 7631.012} C_VEL
LIN {X 0,Y 142.761,Z 1180.582,A -85,B 0,C 180,E1 7621.559,E2 7621.559} C_VEL
LIN {X 0,Y 149.394,Z 1176.992,A -85,B 0,C 180,E1 7613.433,E2 7613.433} C_VEL
LIN {X 0,Y 158.323,Z 1172.373,A -85,B 0,C 180,E1 7605.998,E2 7605.998} C_VEL
LIN {X 0,Y 170.086,Z 1166.314,A -85,B 0,C 180,E1 7598.978,E2 7598.978} C_VEL
LIN {X 0,Y 186.882,Z 1157.389,A -85,B 0,C 180,E1 7591.714,E2 7591.714} C_VEL
LIN {X 0,Y 204.195,Z 1147.42,A -85,B 0,C 180,E1 7586.149,E2 7586.149} C_VEL
LIN {X 0,Y 220.132,Z 1137.631,A -85,B 0,C 180,E1 7582.092,E2 7582.092} C_VEL
LIN {X 0,Y 237.249,Z 1126.321,A -85,B 0,C 180,E1 7578.517,E2 7578.517} C_VEL
LIN {X 0,Y 259.49,Z 1110.127,A -85,B 0,C 180,E1 7574.728,E2 7574.728} C_VEL
LIN {X 0,Y 276.499,Z 1096.435,A -85,B 0,C 180,E1 7572.319,E2 7572.319} C_VEL
LIN {X 0,Y 291.785,Z 1083.077,A -85,B 0,C 180,E1 7570.436,E2 7570.436} C_VEL
LIN {X 0,Y 307.507,Z 1068.139,A -85,B 0,C 180,E1 7568.715,E2 7568.715} C_VEL
LIN {X 0,Y 325.843,Z 1049.039,A -85,B 0,C 180,E1 7566.945,E2 7566.945} C_VEL
LIN {X 0,Y 342.528,Z 1029.375,A -85,B 0,C 180,E1 7565.501,E2 7565.501} C_VEL
LIN {X 0,Y 356.019,Z 1011.861,A -85,B 0,C 180,E1 7564.446,E2 7564.446} C_VEL
LIN {X 0,Y 367.998,Z 994.766,A -85,B 0,C 180,E1 7563.583,E2 7563.583} C_VEL
LIN {X 0,Y 379.889,Z 976.014,A -85,B 0,C 180,E1 7562.772,E2 7562.772} C_VEL
LIN {X 0,Y 393.167,Z 952.556,A -85,B 0,C 180,E1 7561.936,E2 7561.936} C_VEL
LIN {X 0,Y 405.034,Z 927.894,A -85,B 0,C 180,E1 7561.225,E2 7561.225} C_VEL
LIN {X 0,Y 413.475,Z 907.778,A -85,B 0,C 180,E1 7560.746,E2 7560.746} C_VEL
LIN {X 0,Y 420.946,Z 887.245,A -85,B 0,C 180,E1 7560.335,E2 7560.335} C_VEL
LIN {X 0,Y 423.659,Z 879.234,A -85,B 0,C 180,E1 7560.19,E2 7560.19} C_VEL
LIN {X 0,Y 427.29,Z 879.915,A -85,B 0,C 180,E1 7560.006,E2 7560.006} C_VEL
LIN {X 0,Y 427.29,Z 951.419,A -85,B 0,C 180,E1 7560.006,E2 7560.006} C_VEL
LIN {X 0,Y 406.848,Z 951.419,A -85,B 0,C 180,E1 7560.407,E2 7560.407} C_VEL
LIN {X 0,Y 404.869,Z 949.419,A -85,B 0,C 180,E1 7560.448,E2 7560.448} C_VEL
LIN {X 0,Y 404.869,Z 937.144,A -85,B 0,C 180,E1 7560.448,E2 7560.448} C_VEL
LIN {X 0,Y 401.272,Z 936.221,A -85,B 0,C 180,E1 7560.286,E2 7560.286} C_VEL
LIN {X 0,Y 389.601,Z 959.077,A -85,B 0,C 180,E1 7559.706,E2 7559.706} C_VEL
LIN {X 0,Y 378.49,Z 978.419,A -85,B 0,C 180,E1 7559.106,E2 7559.106} C_VEL
LIN {X 0,Y 366.588,Z 997.057,A -85,B 0,C 180,E1 7558.414,E2 7558.414} C_VEL
LIN {X 0,Y 353.268,Z 1015.908,A -85,B 0,C 180,E1 7557.563,E2 7557.563} C_VEL
LIN {X 0,Y 335.155,Z 1038.812,A -85,B 0,C 180,E1 7556.287,E2 7556.287} C_VEL
LIN {X 0,Y 319.158,Z 1056.812,A -85,B 0,C 180,E1 7555.021,E2 7555.021} C_VEL
LIN {X 0,Y 303.819,Z 1072.594,A -85,B 0,C 180,E1 7553.652,E2 7553.652} C_VEL
LIN {X 0,Y 287.738,Z 1087.781,A -85,B 0,C 180,E1 7552.029,E2 7552.029} C_VEL
LIN {X 0,Y 269.157,Z 1103.877,A -85,B 0,C 180,E1 7549.87,E2 7549.87} C_VEL
LIN {X 0,Y 248.057,Z 1120.295,A -85,B 0,C 180,E1 7546.954,E2 7546.954} C_VEL
LIN {X 0,Y 230.818,Z 1132.561,A -85,B 0,C 180,E1 7544.082,E2 7544.082} C_VEL
LIN {X 0,Y 214.811,Z 1143.141,A -85,B 0,C 180,E1 7540.888,E2 7540.888} C_VEL
LIN {X 0,Y 198.766,Z 1153.041,A -85,B 0,C 180,E1 7537.006,E2 7537.006} C_VEL
LIN {X 0,Y 180.168,Z 1163.833,A -85,B 0,C 180,E1 7531.263,E2 7531.263} C_VEL
LIN {X 0,Y 163.035,Z 1173.017,A -85,B 0,C 180,E1 7524.05,E2 7524.05} C_VEL
LIN {X 0,Y 150.74,Z 1179.473,A -85,B 0,C 180,E1 7516.855,E2 7516.855} C_VEL
LIN {X 0,Y 140.984,Z 1184.688,A -85,B 0,C 180,E1 7508.726,E2 7508.726} C_VEL
LIN {X 0,Y 133.585,Z 1188.997,A -85,B 0,C 180,E1 7499.111,E2 7499.111} C_VEL
LIN {X 0,Y 129.018,Z 1192.399,A -85,B 0,C 180,E1 7487.127,E2 7487.127} C_VEL
LIN {X 0,Y 128.068,Z 1193.813,A -85,B 0,C 180,E1 7477.452,E2 7477.452} C_VEL
LIN {X 0,Y 128.08,Z 1194.217,A -85,B 0,C 180,E1 7470,E2 7470} C_VEL
LIN {X 0,Y 128.069,Z 1193.809,A -85,B 0,C 180,E1 7462.548,E2 7462.548} C_VEL
LIN {X 0,Y 129.015,Z 1192.386,A -85,B 0,C 180,E1 7452.873,E2 7452.873} C_VEL
LIN {X 0,Y 133.334,Z 1189.134,A -85,B 0,C 180,E1 7441.319,E2 7441.319} C_VEL
LIN {X 0,Y 140.514,Z 1184.91,A -85,B 0,C 180,E1 7431.752,E2 7431.752} C_VEL
LIN {X 0,Y 150.234,Z 1179.687,A -85,B 0,C 180,E1 7423.495,E2 7423.495} C_VEL
LIN {X 0,Y 161.818,Z 1173.581,A -85,B 0,C 180,E1 7416.558,E2 7416.558} C_VEL
LIN {X 0,Y 177.445,Z 1165.203,A -85,B 0,C 180,E1 7409.728,E2 7409.728} C_VEL
LIN {X 0,Y 197.209,Z 1153.884,A -85,B 0,C 180,E1 7403.412,E2 7403.412} C_VEL
LIN {X 0,Y 213.982,Z 1143.559,A -85,B 0,C 180,E1 7399.288,E2 7399.288} C_VEL
LIN {X 0,Y 229.952,Z 1133.02,A -85,B 0,C 180,E1 7396.069,E2 7396.069} C_VEL
LIN {X 0,Y 247.436,Z 1120.594,A -85,B 0,C 180,E1 7393.133,E2 7393.133} C_VEL
LIN {X 0,Y 268.233,Z 1104.471,A -85,B 0,C 180,E1 7390.239,E2 7390.239} C_VEL
LIN {X 0,Y 287.38,Z 1087.891,A -85,B 0,C 180,E1 7388,E2 7388} C_VEL
LIN {X 0,Y 303.337,Z 1072.827,A -85,B 0,C 180,E1 7386.384,E2 7386.384} C_VEL
LIN {X 0,Y 319.154,Z 1056.55,A -85,B 0,C 180,E1 7384.97,E2 7384.97} C_VEL
LIN {X 0,Y 337.588,Z 1035.649,A -85,B 0,C 180,E1 7383.521,E2 7383.521} C_VEL
LIN {X 0,Y 353.757,Z 1014.864,A -85,B 0,C 180,E1 7382.393,E2 7382.393} C_VEL
LIN {X 0,Y 366.091,Z 997.383,A -85,B 0,C 180,E1 7381.606,E2 7381.606} C_VEL
LIN {X 0,Y 378.012,Z 978.745,A -85,B 0,C 180,E1 7380.909,E2 7380.909} C_VEL
LIN {X 0,Y 389.387,Z 958.96,A -85,B 0,C 180,E1 7380.294,E2 7380.294} C_VEL
LIN {X 0,Y 401.948,Z 934.239,A -85,B 0,C 180,E1 7379.671,E2 7379.671} C_VEL
LIN {X 0,Y 389.543,Z 958.481,A -85,B 0,C 180,E1 7378.97,E2 7378.97} C_VEL
LIN {X 0,Y 378.609,Z 977.391,A -85,B 0,C 180,E1 7378.314,E2 7378.314} C_VEL
LIN {X 0,Y 366.754,Z 995.823,A -85,B 0,C 180,E1 7377.551,E2 7377.551} C_VEL
LIN {X 0,Y 354.041,Z 1013.688,A -85,B 0,C 180,E1 7376.685,E2 7376.685} C_VEL
LIN {X 0,Y 336.992,Z 1035.279,A -85,B 0,C 180,E1 7375.405,E2 7375.405} C_VEL
LIN {X 0,Y 319.245,Z 1055.016,A -85,B 0,C 180,E1 7373.927,E2 7373.927} C_VEL
LIN {X 0,Y 304.527,Z 1069.935,A -85,B 0,C 180,E1 7372.549,E2 7372.549} C_VEL
LIN {X 0,Y 289.529,Z 1083.9,A -85,B 0,C 180,E1 7370.992,E2 7370.992} C_VEL
LIN {X 0,Y 272.932,Z 1098.093,A -85,B 0,C 180,E1 7369.048,E2 7369.048} C_VEL
LIN {X 0,Y 252.246,Z 1114.205,A -85,B 0,C 180,E1 7366.199,E2 7366.199} C_VEL
LIN {X 0,Y 233.109,Z 1127.523,A -85,B 0,C 180,E1 7363.037,E2 7363.037} C_VEL
LIN {X 0,Y 216.402,Z 1138.232,A -85,B 0,C 180,E1 7359.707,E2 7359.707} C_VEL
LIN {X 0,Y 200.442,Z 1147.707,A -85,B 0,C 180,E1 7355.855,E2 7355.855} C_VEL
LIN {X 0,Y 181.321,Z 1158.289,A -85,B 0,C 180,E1 7349.968,E2 7349.968} C_VEL
LIN {X 0,Y 164.303,Z 1166.836,A -85,B 0,C 180,E1 7342.863,E2 7342.863} C_VEL
LIN {X 0,Y 152.537,Z 1172.549,A -85,B 0,C 180,E1 7336.14,E2 7336.14} C_VEL
LIN {X 0,Y 142.491,Z 1177.385,A -85,B 0,C 180,E1 7328.133,E2 7328.133} C_VEL
LIN {X 0,Y 134.544,Z 1181.396,A -85,B 0,C 180,E1 7318.399,E2 7318.399} C_VEL
LIN {X 0,Y 129.569,Z 1184.325,A -85,B 0,C 180,E1 7306.59,E2 7306.59} C_VEL
LIN {X 0,Y 128.244,Z 1185.476,A -85,B 0,C 180,E1 7297.166,E2 7297.166} C_VEL
LIN {X 0,Y 128.079,Z 1185.798,A -85,B 0,C 180,E1 7289.553,E2 7289.553} C_VEL
LIN {X 0,Y 128.331,Z 1185.427,A -85,B 0,C 180,E1 7281.487,E2 7281.487} C_VEL
LIN {X 0,Y 130.169,Z 1183.967,A -85,B 0,C 180,E1 7271.179,E2 7271.179} C_VEL
LIN {X 0,Y 135.303,Z 1181.003,A -85,B 0,C 180,E1 7260.323,E2 7260.323} C_VEL
LIN {X 0,Y 142.822,Z 1177.266,A -85,B 0,C 180,E1 7251.46,E2 7251.46} C_VEL
LIN {X 0,Y 152.453,Z 1172.645,A -85,B 0,C 180,E1 7243.827,E2 7243.827} C_VEL
LIN {X 0,Y 164.824,Z 1166.657,A -85,B 0,C 180,E1 7236.799,E2 7236.799} C_VEL
LIN {X 0,Y 182.636,Z 1157.662,A -85,B 0,C 180,E1 7229.488,E2 7229.488} C_VEL
LIN {X 0,Y 200.403,Z 1147.837,A -85,B 0,C 180,E1 7224.073,E2 7224.073} C_VEL
LIN {X 0,Y 216.312,Z 1138.407,A -85,B 0,C 180,E1 7220.229,E2 7220.229} C_VEL
LIN {X 0,Y 233.027,Z 1127.716,A -85,B 0,C 180,E1 7216.896,E2 7216.896} C_VEL
LIN {X 0,Y 253.058,Z 1113.796,A -85,B 0,C 180,E1 7213.598,E2 7213.598} C_VEL
LIN {X 0,Y 272.866,Z 1098.351,A -85,B 0,C 180,E1 7210.881,E2 7210.881} C_VEL
LIN {X 0,Y 289.47,Z 1084.178,A -85,B 0,C 180,E1 7208.934,E2 7208.934} C_VEL
LIN {X 0,Y 304.726,Z 1069.993,A -85,B 0,C 180,E1 7207.352,E2 7207.352} C_VEL
LIN {X 0,Y 320.637,Z 1053.837,A -85,B 0,C 180,E1 7205.873,E2 7205.873} C_VEL
LIN {X 0,Y 339.334,Z 1032.755,A -85,B 0,C 180,E1 7204.332,E2 7204.332} C_VEL
LIN {X 0,Y 354.911,Z 1012.895,A -85,B 0,C 180,E1 7203.175,E2 7203.175} C_VEL
LIN {X 0,Y 367.253,Z 995.512,A -85,B 0,C 180,E1 7202.34,E2 7202.34} C_VEL
LIN {X 0,Y 379.089,Z 977.081,A -85,B 0,C 180,E1 7201.58,E2 7201.58} C_VEL
LIN {X 0,Y 390.988,Z 956.397,A -85,B 0,C 180,E1 7200.87,E2 7200.87} C_VEL
LIN {X 0,Y 401.272,Z 936.221,A -85,B 0,C 180,E1 7200.286,E2 7200.286} C_VEL
LIN {X 0,Y 404.669,Z 937.188,A -85,B 0,C 180,E1 7200.06,E2 7200.06} C_VEL
LIN {X 0,Y 404.669,Z 991.117,A -85,B 0,C 180,E1 7200.06,E2 7200.06} C_VEL
LIN {X 0,Y 384.17,Z 991.117,A -85,B 0,C 180,E1 7200.521,E2 7200.521} C_VEL
LIN {X 0,Y 382.195,Z 989.117,A -85,B 0,C 180,E1 7200.568,E2 7200.568} C_VEL
LIN {X 0,Y 382.195,Z 978.711,A -85,B 0,C 180,E1 7200.568,E2 7200.568} C_VEL
LIN {X 0,Y 378.787,Z 977.609,A -85,B 0,C 180,E1 7200.364,E2 7200.364} C_VEL
LIN {X 0,Y 366.951,Z 996.053,A -85,B 0,C 180,E1 7199.723,E2 7199.723} C_VEL
LIN {X 0,Y 354.007,Z 1014.295,A -85,B 0,C 180,E1 7198.96,E2 7198.96} C_VEL
LIN {X 0,Y 336.691,Z 1036.298,A -85,B 0,C 180,E1 7197.837,E2 7197.837} C_VEL
LIN {X 0,Y 318.545,Z 1056.543,A -85,B 0,C 180,E1 7196.509,E2 7196.509} C_VEL
LIN {X 0,Y 303.011,Z 1072.324,A -85,B 0,C 180,E1 7195.216,E2 7195.216} C_VEL
LIN {X 0,Y 287.653,Z 1086.652,A -85,B 0,C 180,E1 7193.779,E2 7193.779} C_VEL
LIN {X 0,Y 270.616,Z 1101.256,A -85,B 0,C 180,E1 7191.968,E2 7191.968} C_VEL
LIN {X 0,Y 248.399,Z 1118.526,A -85,B 0,C 180,E1 7189.158,E2 7189.158} C_VEL
LIN {X 0,Y 229.53,Z 1131.701,A -85,B 0,C 180,E1 7186.266,E2 7186.266} C_VEL
LIN {X 0,Y 212.192,Z 1142.866,A -85,B 0,C 180,E1 7183.046,E2 7183.046} C_VEL
LIN {X 0,Y 194.811,Z 1153.235,A -85,B 0,C 180,E1 7179.084,E2 7179.084} C_VEL
LIN {X 0,Y 174.549,Z 1164.434,A -85,B 0,C 180,E1 7173.093,E2 7173.093} C_VEL
LIN {X 0,Y 157.587,Z 1173.055,A -85,B 0,C 180,E1 7166.218,E2 7166.218} C_VEL
LIN {X 0,Y 145.118,Z 1179.198,A -85,B 0,C 180,E1 7159.279,E2 7159.279} C_VEL
LIN {X 0,Y 134.897,Z 1184.244,A -85,B 0,C 180,E1 7151.275,E2 7151.275} C_VEL
LIN {X 0,Y 126.842,Z 1188.464,A -85,B 0,C 180,E1 7141.64,E2 7141.64} C_VEL
LIN {X 0,Y 121.461,Z 1191.979,A -85,B 0,C 180,E1 7129.225,E2 7129.225} C_VEL
LIN {X 0,Y 120.094,Z 1193.511,A -85,B 0,C 180,E1 7118.619,E2 7118.619} C_VEL
LIN {X 0,Y 120.078,Z 1193.917,A -85,B 0,C 180,E1 7110.954,E2 7110.954} C_VEL
LIN {X 0,Y 120.054,Z 1193.64,A -85,B 0,C 180,E1 7103.784,E2 7103.784} C_VEL
LIN {X 0,Y 120.467,Z 1192.789,A -85,B 0,C 180,E1 7096.072,E2 7096.072} C_VEL
LIN {X 0,Y 122.602,Z 1190.999,A -85,B 0,C 180,E1 7086.955,E2 7086.955} C_VEL
LIN {X 0,Y 127.564,Z 1188.018,A -85,B 0,C 180,E1 7077.26,E2 7077.26} C_VEL
LIN {X 0,Y 135.432,Z 1183.931,A -85,B 0,C 180,E1 7068.218,E2 7068.218} C_VEL
LIN {X 0,Y 146.243,Z 1178.6,A -85,B 0,C 180,E1 7059.993,E2 7059.993} C_VEL
LIN {X 0,Y 162.831,Z 1170.436,A -85,B 0,C 180,E1 7051.403,E2 7051.403} C_VEL
LIN {X 0,Y 180.832,Z 1160.919,A -85,B 0,C 180,E1 7044.849,E2 7044.849} C_VEL
LIN {X 0,Y 197.225,Z 1151.723,A -85,B 0,C 180,E1 7040.302,E2 7040.302} C_VEL
LIN {X 0,Y 214.157,Z 1141.532,A -85,B 0,C 180,E1 7036.547,E2 7036.547} C_VEL
LIN {X 0,Y 235.432,Z 1127.659,A -85,B 0,C 180,E1 7032.759,E2 7032.759} C_VEL
LIN {X 0,Y 255.723,Z 1112.826,A -85,B 0,C 180,E1 7029.837,E2 7029.837} C_VEL
LIN {X 0,Y 272.557,Z 1099.439,A -85,B 0,C 180,E1 7027.801,E2 7027.801} C_VEL
LIN {X 0,Y 288.602,Z 1085.577,A -85,B 0,C 180,E1 7026.118,E2 7026.118} C_VEL
LIN {X 0,Y 304.942,Z 1070.207,A -85,B 0,C 180,E1 7024.609,E2 7024.609} C_VEL
LIN {X 0,Y 324.409,Z 1050.023,A -85,B 0,C 180,E1 7023.039,E2 7023.039} C_VEL
LIN {X 0,Y 341.621,Z 1029.843,A -85,B 0,C 180,E1 7021.814,E2 7021.814} C_VEL
LIN {X 0,Y 355.496,Z 1011.894,A -85,B 0,C 180,E1 7020.937,E2 7020.937} C_VEL
LIN {X 0,Y 368.449,Z 993.406,A -85,B 0,C 180,E1 7020.182,E2 7020.182} C_VEL
LIN {X 0,Y 379.406,Z 976.132,A -85,B 0,C 180,E1 7019.595,E2 7019.595} C_VEL
LIN {X 0,Y 367.517,Z 994.597,A -85,B 0,C 180,E1 7018.883,E2 7018.883} C_VEL
LIN {X 0,Y 355.143,Z 1011.976,A -85,B 0,C 180,E1 7018.103,E2 7018.103} C_VEL
LIN {X 0,Y 341.248,Z 1029.68,A -85,B 0,C 180,E1 7017.145,E2 7017.145} C_VEL
LIN {X 0,Y 323.33,Z 1050.28,A -85,B 0,C 180,E1 7015.78,E2 7015.78} C_VEL
LIN {X 0,Y 305.485,Z 1068.381,A -85,B 0,C 180,E1 7014.264,E2 7014.264} C_VEL
LIN {X 0,Y 289.296,Z 1083.341,A -85,B 0,C 180,E1 7012.711,E2 7012.711} C_VEL
LIN {X 0,Y 272.96,Z 1097.161,A -85,B 0,C 180,E1 7010.937,E2 7010.937} C_VEL
LIN {X 0,Y 254.017,Z 1111.814,A -85,B 0,C 180,E1 7008.552,E2 7008.552} C_VEL
LIN {X 0,Y 231.692,Z 1127.237,A -85,B 0,C 180,E1 7005.163,E2 7005.163} C_VEL
LIN {X 0,Y 214.492,Z 1138.005,A -85,B 0,C 180,E1 7001.979,E2 7001.979} C_VEL
LIN {X 0,Y 198.026,Z 1147.505,A -85,B 0,C 180,E1 6998.285,E2 6998.285} C_VEL
LIN {X 0,Y 180.989,Z 1156.606,A -85,B 0,C 180,E1 6993.502,E2 6993.502} C_VEL
LIN {X 0,Y 160.698,Z 1166.525,A -85,B 0,C 180,E1 6985.845,E2 6985.845} C_VEL
LIN {X 0,Y 147.449,Z 1172.579,A -85,B 0,C 180,E1 6978.824,E2 6978.824} C_VEL
LIN {X 0,Y 136.509,Z 1177.46,A -85,B 0,C 180,E1 6970.683,E2 6970.683} C_VEL
LIN {X 0,Y 128.268,Z 1181.212,A -85,B 0,C 180,E1 6961.485,E2 6961.485} C_VEL
LIN {X 0,Y 122.585,Z 1184.138,A -85,B 0,C 180,E1 6950.277,E2 6950.277} C_VEL
LIN {X 0,Y 120.384,Z 1185.683,A -85,B 0,C 180,E1 6939.08,E2 6939.08} C_VEL
LIN {X 0,Y 120.085,Z 1186.052,A -85,B 0,C 180,E1 6930.477,E2 6930.477} C_VEL
LIN {X 0,Y 120.27,Z 1185.749,A -85,B 0,C 180,E1 6922.356,E2 6922.356} C_VEL
LIN {X 0,Y 121.813,Z 1184.604,A -85,B 0,C 180,E1 6912.209,E2 6912.209} C_VEL
LIN {X 0,Y 127.432,Z 1181.672,A -85,B 0,C 180,E1 6899.668,E2 6899.668} C_VEL
LIN {X 0,Y 136.005,Z 1177.735,A -85,B 0,C 180,E1 6889.689,E2 6889.689} C_VEL
LIN {X 0,Y 146.816,Z 1172.917,A -85,B 0,C 180,E1 6881.485,E2 6881.485} C_VEL
LIN {X 0,Y 159.964,Z 1166.93,A -85,B 0,C 180,E1 6874.405,E2 6874.405} C_VEL
LIN {X 0,Y 178.679,Z 1157.934,A -85,B 0,C 180,E1 6867.16,E2 6867.16} C_VEL
LIN {X 0,Y 197.142,Z 1148.11,A -85,B 0,C 180,E1 6861.855,E2 6861.855} C_VEL
LIN {X 0,Y 213.57,Z 1138.679,A -85,B 0,C 180,E1 6858.127,E2 6858.127} C_VEL
LIN {X 0,Y 230.743,Z 1127.988,A -85,B 0,C 180,E1 6854.916,E2 6854.916} C_VEL
LIN {X 0,Y 251.718,Z 1113.73,A -85,B 0,C 180,E1 6851.688,E2 6851.688} C_VEL
LIN {X 0,Y 272.354,Z 1097.862,A -85,B 0,C 180,E1 6849.053,E2 6849.053} C_VEL
LIN {X 0,Y 288.302,Z 1084.447,A -85,B 0,C 180,E1 6847.311,E2 6847.311} C_VEL
LIN {X 0,Y 304.487,Z 1069.588,A -85,B 0,C 180,E1 6845.748,E2 6845.748} C_VEL
LIN {X 0,Y 321.558,Z 1052.391,A -85,B 0,C 180,E1 6844.28,E2 6844.28} C_VEL
LIN {X 0,Y 340.369,Z 1031.108,A -85,B 0,C 180,E1 6842.84,E2 6842.84} C_VEL
LIN {X 0,Y 354.634,Z 1013.049,A -85,B 0,C 180,E1 6841.854,E2 6841.854} C_VEL
LIN {X 0,Y 367.516,Z 995.032,A -85,B 0,C 180,E1 6841.041,E2 6841.041} C_VEL
LIN {X 0,Y 378.787,Z 977.609,A -85,B 0,C 180,E1 6840.364,E2 6840.364} C_VEL
LIN {X 0,Y 382.217,Z 978.713,A -85,B 0,C 180,E1 6840.168,E2 6840.168} C_VEL
LIN {X 0,Y 382.217,Z 1023.059,A -85,B 0,C 180,E1 6840.168,E2 6840.168} C_VEL
LIN {X 0,Y 361.636,Z 1023.059,A -85,B 0,C 180,E1 6840.574,E2 6840.574} C_VEL
LIN {X 0,Y 359.653,Z 1021.059,A -85,B 0,C 180,E1 6840.616,E2 6840.616} C_VEL
LIN {X 0,Y 359.653,Z 1012.131,A -85,B 0,C 180,E1 6840.616,E2 6840.616} C_VEL
LIN {X 0,Y 356.287,Z 1010.891,A -85,B 0,C 180,E1 6840.425,E2 6840.425} C_VEL
LIN {X 0,Y 342.458,Z 1028.686,A -85,B 0,C 180,E1 6839.621,E2 6839.621} C_VEL
LIN {X 0,Y 327.543,Z 1046.127,A -85,B 0,C 180,E1 6838.652,E2 6838.652} C_VEL
LIN {X 0,Y 308.31,Z 1066.429,A -85,B 0,C 180,E1 6837.251,E2 6837.251} C_VEL
LIN {X 0,Y 289.771,Z 1083.809,A -85,B 0,C 180,E1 6835.706,E2 6835.706} C_VEL
LIN {X 0,Y 273.233,Z 1097.983,A -85,B 0,C 180,E1 6834.119,E2 6834.119} C_VEL
LIN {X 0,Y 256.308,Z 1111.3,A -85,B 0,C 180,E1 6832.244,E2 6832.244} C_VEL
LIN {X 0,Y 237.678,Z 1124.738,A -85,B 0,C 180,E1 6829.823,E2 6829.823} C_VEL
LIN {X 0,Y 214.268,Z 1139.956,A -85,B 0,C 180,E1 6826.074,E2 6826.074} C_VEL
LIN {X 0,Y 195.294,Z 1151.075,A -85,B 0,C 180,E1 6822.227,E2 6822.227} C_VEL
LIN {X 0,Y 178.635,Z 1160.105,A -85,B 0,C 180,E1 6817.974,E2 6817.974} C_VEL
LIN {X 0,Y 161.466,Z 1168.78,A -85,B 0,C 180,E1 6812.314,E2 6812.314} C_VEL
LIN {X 0,Y 142.061,Z 1177.902,A -85,B 0,C 180,E1 6803.254,E2 6803.254} C_VEL
LIN {X 0,Y 129.665,Z 1183.536,A -85,B 0,C 180,E1 6794.564,E2 6794.564} C_VEL
LIN {X 0,Y 120.994,Z 1187.609,A -85,B 0,C 180,E1 6785.342,E2 6785.342} C_VEL
LIN {X 0,Y 115.471,Z 1190.508,A -85,B 0,C 180,E1 6775.655,E2 6775.655} C_VEL
LIN {X 0,Y 112.74,Z 1192.387,A -85,B 0,C 180,E1 6765.958,E2 6765.958} C_VEL
LIN {X 0,Y 112.069,Z 1193.354,A -85,B 0,C 180,E1 6757.175,E2 6757.175} C_VEL
LIN {X 0,Y 112.081,Z 1193.674,A -85,B 0,C 180,E1 6749.489,E2 6749.489} C_VEL
LIN {X 0,Y 112.099,Z 1193.269,A -85,B 0,C 180,E1 6741.279,E2 6741.279} C_VEL
LIN {X 0,Y 113.751,Z 1191.692,A -85,B 0,C 180,E1 6729.415,E2 6729.415} C_VEL
LIN {X 0,Y 119.672,Z 1188.251,A -85,B 0,C 180,E1 6716.535,E2 6716.535} C_VEL
LIN {X 0,Y 128.255,Z 1184.143,A -85,B 0,C 180,E1 6706.683,E2 6706.683} C_VEL
LIN {X 0,Y 139.772,Z 1178.869,A -85,B 0,C 180,E1 6698.105,E2 6698.105} C_VEL
LIN {X 0,Y 153.729,Z 1172.397,A -85,B 0,C 180,E1 6690.848,E2 6690.848} C_VEL
LIN {X 0,Y 173.45,Z 1162.771,A -85,B 0,C 180,E1 6683.572,E2 6683.572} C_VEL
LIN {X 0,Y 192.778,Z 1152.385,A -85,B 0,C 180,E1 6678.352,E2 6678.352} C_VEL
LIN {X 0,Y 209.876,Z 1142.474,A -85,B 0,C 180,E1 6674.739,E2 6674.739} C_VEL
LIN {X 0,Y 227.742,Z 1131.244,A -85,B 0,C 180,E1 6671.652,E2 6671.652} C_VEL
LIN {X 0,Y 249.743,Z 1116.113,A -85,B 0,C 180,E1 6668.556,E2 6668.556} C_VEL
LIN {X 0,Y 270.556,Z 1099.973,A -85,B 0,C 180,E1 6666.153,E2 6666.153} C_VEL
LIN {X 0,Y 286.863,Z 1086.158,A -85,B 0,C 180,E1 6664.553,E2 6664.553} C_VEL
LIN {X 0,Y 302.429,Z 1071.806,A -85,B 0,C 180,E1 6663.204,E2 6663.204} C_VEL
LIN {X 0,Y 318.292,Z 1055.847,A -85,B 0,C 180,E1 6661.98,E2 6661.98} C_VEL
LIN {X 0,Y 336.977,Z 1035.098,A -85,B 0,C 180,E1 6660.714,E2 6660.714} C_VEL
LIN {X 0,Y 353.453,Z 1014.315,A -85,B 0,C 180,E1 6659.726,E2 6659.726} C_VEL
LIN {X 0,Y 356.801,Z 1009.812,A -85,B 0,C 180,E1 6659.528,E2 6659.528} C_VEL
LIN {X 0,Y 343.045,Z 1027.39,A -85,B 0,C 180,E1 6658.653,E2 6658.653} C_VEL
LIN {X 0,Y 329.216,Z 1043.463,A -85,B 0,C 180,E1 6657.708,E2 6657.708} C_VEL
LIN {X 0,Y 313.091,Z 1060.518,A -85,B 0,C 180,E1 6656.491,E2 6656.491} C_VEL
LIN {X 0,Y 291.246,Z 1081.116,A -85,B 0,C 180,E1 6654.61,E2 6654.61} C_VEL
LIN {X 0,Y 273.707,Z 1095.891,A -85,B 0,C 180,E1 6652.865,E2 6652.865} C_VEL
LIN {X 0,Y 257.148,Z 1108.644,A -85,B 0,C 180,E1 6650.973,E2 6650.973} C_VEL
LIN {X 0,Y 239.647,Z 1120.986,A -85,B 0,C 180,E1 6648.657,E2 6648.657} C_VEL
LIN {X 0,Y 218.174,Z 1134.757,A -85,B 0,C 180,E1 6645.234,E2 6645.234} C_VEL
LIN {X 0,Y 197.361,Z 1146.562,A -85,B 0,C 180,E1 6641.08,E2 6641.08} C_VEL
LIN {X 0,Y 180.538,Z 1155.307,A -85,B 0,C 180,E1 6636.83,E2 6636.83} C_VEL
LIN {X 0,Y 164.632,Z 1162.95,A -85,B 0,C 180,E1 6631.718,E2 6631.718} C_VEL
LIN {X 0,Y 146.989,Z 1170.891,A -85,B 0,C 180,E1 6624.044,E2 6624.044} C_VEL
LIN {X 0,Y 132.288,Z 1176.945,A -85,B 0,C 180,E1 6614.661,E2 6614.661} C_VEL
LIN {X 0,Y 122.738,Z 1180.877,A -85,B 0,C 180,E1 6605.337,E2 6605.337} C_VEL
LIN {X 0,Y 116.497,Z 1183.605,A -85,B 0,C 180,E1 6595.413,E2 6595.413} C_VEL
LIN {X 0,Y 113.328,Z 1185.231,A -85,B 0,C 180,E1 6585.873,E2 6585.873} C_VEL
LIN {X 0,Y 112.246,Z 1186.043,A -85,B 0,C 180,E1 6577.164,E2 6577.164} C_VEL
LIN {X 0,Y 112.088,Z 1186.3,A -85,B 0,C 180,E1 6568.978,E2 6568.978} C_VEL
LIN {X 0,Y 112.48,Z 1185.936,A -85,B 0,C 180,E1 6559.759,E2 6559.759} C_VEL
LIN {X 0,Y 115.219,Z 1184.288,A -85,B 0,C 180,E1 6547.553,E2 6547.553} C_VEL
LIN {X 0,Y 121.42,Z 1181.479,A -85,B 0,C 180,E1 6536.278,E2 6536.278} C_VEL
LIN {X 0,Y 130.27,Z 1177.809,A -85,B 0,C 180,E1 6526.914,E2 6526.914} C_VEL
LIN {X 0,Y 141.442,Z 1173.189,A -85,B 0,C 180,E1 6518.959,E2 6518.959} C_VEL
LIN {X 0,Y 155.502,Z 1167.159,A -85,B 0,C 180,E1 6511.821,E2 6511.821} C_VEL
LIN {X 0,Y 175.025,Z 1158.207,A -85,B 0,C 180,E1 6504.728,E2 6504.728} C_VEL
LIN {X 0,Y 194.285,Z 1148.33,A -85,B 0,C 180,E1 6499.544,E2 6499.544} C_VEL
LIN {X 0,Y 211.396,Z 1138.793,A -85,B 0,C 180,E1 6495.923,E2 6495.923} C_VEL
LIN {X 0,Y 228.919,Z 1128.147,A -85,B 0,C 180,E1 6492.871,E2 6492.871} C_VEL
LIN {X 0,Y 250.598,Z 1113.692,A -85,B 0,C 180,E1 6489.769,E2 6489.769} C_VEL
LIN {X 0,Y 271.175,Z 1098.131,A -85,B 0,C 180,E1 6487.326,E2 6487.326} C_VEL
LIN {X 0,Y 287.368,Z 1084.716,A -85,B 0,C 180,E1 6485.677,E2 6485.677} C_VEL
LIN {X 0,Y 303.772,Z 1069.855,A -85,B 0,C 180,E1 6484.202,E2 6484.202} C_VEL
LIN {X 0,Y 320.499,Z 1053.22,A -85,B 0,C 180,E1 6482.861,E2 6482.861} C_VEL
LIN {X 0,Y 340.062,Z 1031.373,A -85,B 0,C 180,E1 6481.466,E2 6481.466} C_VEL
LIN {X 0,Y 354.464,Z 1013.312,A -85,B 0,C 180,E1 6480.537,E2 6480.537} C_VEL
LIN {X 0,Y 356.287,Z 1010.891,A -85,B 0,C 180,E1 6480.425,E2 6480.425} C_VEL
LIN {X 0,Y 349.506,Z 1019.978,A -85,B 0,C 180,E1 6480.194,E2 6480.194} C_VEL
LIN {X 0,Y 341.432,Z 1029.808,A -85,B 0,C 180,E1 6480.243,E2 6480.243} C_VEL
LIN {X 0,Y 332.172,Z 1040.57,A -85,B 0,C 180,E1 6480.61,E2 6480.61} C_VEL
LIN {X 0,Y 325.793,Z 1047.589,A -85,B 0,C 180,E1 6481.008,E2 6481.008} C_VEL
LIN {X 0,Y 305.245,Z 1068.295,A -85,B 0,C 180,E1 6482.496,E2 6482.496} C_VEL
LIN {X 0,Y 288.613,Z 1083.317,A -85,B 0,C 180,E1 6483.862,E2 6483.862} C_VEL
LIN {X 0,Y 272.166,Z 1096.883,A -85,B 0,C 180,E1 6485.396,E2 6485.396} C_VEL
LIN {X 0,Y 254.989,Z 1109.83,A -85,B 0,C 180,E1 6487.226,E2 6487.226} C_VEL
LIN {X 0,Y 233.471,Z 1124.578,A -85,B 0,C 180,E1 6489.94,E2 6489.94} C_VEL
LIN {X 0,Y 211.656,Z 1137.713,A -85,B 0,C 180,E1 6493.31,E2 6493.31} C_VEL
LIN {X 0,Y 193.265,Z 1147.76,A -85,B 0,C 180,E1 6496.844,E2 6496.844} C_VEL
LIN {X 0,Y 175.716,Z 1156.51,A -85,B 0,C 180,E1 6501.063,E2 6501.063} C_VEL
LIN {X 0,Y 155.065,Z 1165.907,A -85,B 0,C 180,E1 6507.663,E2 6507.663} C_VEL
LIN {X 0,Y 137.627,Z 1172.973,A -85,B 0,C 180,E1 6515.543,E2 6515.543} C_VEL
LIN {X 0,Y 124.865,Z 1177.883,A -85,B 0,C 180,E1 6523.89,E2 6523.89} C_VEL
LIN {X 0,Y 115.262,Z 1181.51,A -85,B 0,C 180,E1 6533.234,E2 6533.234} C_VEL
LIN {X 0,Y 108.622,Z 1184.13,A -85,B 0,C 180,E1 6543.779,E2 6543.779} C_VEL
LIN {X 0,Y 105.19,Z 1185.711,A -85,B 0,C 180,E1 6554.565,E2 6554.565} C_VEL
LIN {X 0,Y 104.211,Z 1186.354,A -85,B 0,C 180,E1 6563.389,E2 6563.389} C_VEL
LIN {X 0,Y 104.095,Z 1186.532,A -85,B 0,C 180,E1 6571.651,E2 6571.651} C_VEL
LIN {X 0,Y 104.629,Z 1186.126,A -85,B 0,C 180,E1 6581.577,E2 6581.577} C_VEL
LIN {X 0,Y 107.963,Z 1184.406,A -85,B 0,C 180,E1 6594.629,E2 6594.629} C_VEL
LIN {X 0,Y 114.549,Z 1181.753,A -85,B 0,C 180,E1 6605.79,E2 6605.79} C_VEL
LIN {X 0,Y 124.41,Z 1178.006,A -85,B 0,C 180,E1 6615.666,E2 6615.666} C_VEL
LIN {X 0,Y 137.071,Z 1173.126,A -85,B 0,C 180,E1 6624.065,E2 6624.065} C_VEL
LIN {X 0,Y 154.144,Z 1166.197,A -85,B 0,C 180,E1 6631.904,E2 6631.904} C_VEL
LIN {X 0,Y 174.982,Z 1156.763,A -85,B 0,C 180,E1 6638.652,E2 6638.652} C_VEL
LIN {X 0,Y 192.478,Z 1148.056,A -85,B 0,C 180,E1 6642.904,E2 6642.904} C_VEL
LIN {X 0,Y 209.935,Z 1138.555,A -85,B 0,C 180,E1 6646.309,E2 6646.309} C_VEL
LIN {X 0,Y 228.917,Z 1127.225,A -85,B 0,C 180,E1 6649.342,E2 6649.342} C_VEL
LIN {X 0,Y 252.196,Z 1111.674,A -85,B 0,C 180,E1 6652.372,E2 6652.372} C_VEL
LIN {X 0,Y 270.28,Z 1098.157,A -85,B 0,C 180,E1 6654.338,E2 6654.338} C_VEL
LIN {X 0,Y 286.696,Z 1084.722,A -85,B 0,C 180,E1 6655.889,E2 6655.889} C_VEL
LIN {X 0,Y 302.318,Z 1070.754,A -85,B 0,C 180,E1 6657.195,E2 6657.195} C_VEL
LIN {X 0,Y 318.081,Z 1055.333,A -85,B 0,C 180,E1 6658.379,E2 6658.379} C_VEL
LIN {X 0,Y 334.066,Z 1038.137,A -85,B 0,C 180,E1 6659.48,E2 6659.48} C_VEL
LIN {X 0,Y 316.969,Z 1056.748,A -85,B 0,C 180,E1 6660.563,E2 6660.563} C_VEL
LIN {X 0,Y 300.95,Z 1072.6,A -85,B 0,C 180,E1 6661.714,E2 6661.714} C_VEL
LIN {X 0,Y 284.363,Z 1087.595,A -85,B 0,C 180,E1 6663.055,E2 6663.055} C_VEL
LIN {X 0,Y 262.991,Z 1105.145,A -85,B 0,C 180,E1 6665.071,E2 6665.071} C_VEL
LIN {X 0,Y 242.002,Z 1120.406,A -85,B 0,C 180,E1 6667.439,E2 6667.439} C_VEL
LIN {X 0,Y 224.267,Z 1132.183,A -85,B 0,C 180,E1 6669.84,E2 6669.84} C_VEL
LIN {X 0,Y 206.096,Z 1143.248,A -85,B 0,C 180,E1 6672.805,E2 6672.805} C_VEL
LIN {X 0,Y 184.312,Z 1155.397,A -85,B 0,C 180,E1 6677.299,E2 6677.299} C_VEL
LIN {X 0,Y 163.091,Z 1165.867,A -85,B 0,C 180,E1 6683.133,E2 6683.133} C_VEL
LIN {X 0,Y 147.434,Z 1173.062,A -85,B 0,C 180,E1 6688.974,E2 6688.974} C_VEL
LIN {X 0,Y 133.502,Z 1179.122,A -85,B 0,C 180,E1 6696.015,E2 6696.015} C_VEL
LIN {X 0,Y 120.639,Z 1184.599,A -85,B 0,C 180,E1 6705.463,E2 6705.463} C_VEL
LIN {X 0,Y 109.644,Z 1189.48,A -85,B 0,C 180,E1 6719.291,E2 6719.291} C_VEL
LIN {X 0,Y 105.256,Z 1191.88,A -85,B 0,C 180,E1 6731.157,E2 6731.157} C_VEL
LIN {X 0,Y 104.095,Z 1193.058,A -85,B 0,C 180,E1 6741.716,E2 6741.716} C_VEL
LIN {X 0,Y 104.091,Z 1193.43,A -85,B 0,C 180,E1 6750,E2 6750} C_VEL
LIN {X 0,Y 104.095,Z 1193.059,A -85,B 0,C 180,E1 6758.36,E2 6758.36} C_VEL
LIN {X 0,Y 105.517,Z 1191.745,A -85,B 0,C 180,E1 6769.946,E2 6769.946} C_VEL
LIN {X 0,Y 111.802,Z 1188.519,A -85,B 0,C 180,E1 6784.292,E2 6784.292} C_VEL
LIN {X 0,Y 121.8,Z 1184.129,A -85,B 0,C 180,E1 6795.576,E2 6795.576} C_VEL
LIN {X 0,Y 134.123,Z 1178.912,A -85,B 0,C 180,E1 6804.347,E2 6804.347} C_VEL
LIN {X 0,Y 148.858,Z 1172.502,A -85,B 0,C 180,E1 6811.631,E2 6811.631} C_VEL
LIN {X 0,Y 168.643,Z 1163.399,A -85,B 0,C 180,E1 6818.564,E2 6818.564} C_VEL
LIN {X 0,Y 189.428,Z 1152.682,A -85,B 0,C 180,E1 6823.873,E2 6823.873} C_VEL
LIN {X 0,Y 207.89,Z 1142.314,A -85,B 0,C 180,E1 6827.511,E2 6827.511} C_VEL
LIN {X 0,Y 226.117,Z 1131.15,A -85,B 0,C 180,E1 6830.426,E2 6830.426} C_VEL
LIN {X 0,Y 248.067,Z 1116.422,A -85,B 0,C 180,E1 6833.287,E2 6833.287} C_VEL
LIN {X 0,Y 269.754,Z 1099.928,A -85,B 0,C 180,E1 6835.606,E2 6835.606} C_VEL
LIN {X 0,Y 286.323,Z 1086.109,A -85,B 0,C 180,E1 6837.107,E2 6837.107} C_VEL
LIN {X 0,Y 302.586,Z 1071.303,A -85,B 0,C 180,E1 6838.4,E2 6838.4} C_VEL
LIN {X 0,Y 318.963,Z 1054.98,A -85,B 0,C 180,E1 6839.558,E2 6839.558} C_VEL
LIN {X 0,Y 333.596,Z 1038.979,A -85,B 0,C 180,E1 6840.488,E2 6840.488} C_VEL
LIN {X 0,Y 325.793,Z 1047.589,A -85,B 0,C 180,E1 6841.008,E2 6841.008} C_VEL
LIN {X 0,Y 321.294,Z 1052.446,A -85,B 0,C 180,E1 6841.153,E2 6841.153} C_VEL
LIN {X 0,Y 315.084,Z 1058.806,A -85,B 0,C 180,E1 6840.963,E2 6840.963} C_VEL
LIN {X 0,Y 300.78,Z 1072.617,A -85,B 0,C 180,E1 6839.859,E2 6839.859} C_VEL
LIN {X 0,Y 283.051,Z 1088.409,A -85,B 0,C 180,E1 6838.541,E2 6838.541} C_VEL
LIN {X 0,Y 259.428,Z 1107.212,A -85,B 0,C 180,E1 6836.464,E2 6836.464} C_VEL
LIN {X 0,Y 240.908,Z 1120.392,A -85,B 0,C 180,E1 6834.522,E2 6834.522} C_VEL
LIN {X 0,Y 222.755,Z 1132.187,A -85,B 0,C 180,E1 6832.261,E2 6832.261} C_VEL
LIN {X 0,Y 204.392,Z 1143.091,A -85,B 0,C 180,E1 6829.502,E2 6829.502} C_VEL
LIN {X 0,Y 181.978,Z 1155.221,A -85,B 0,C 180,E1 6825.242,E2 6825.242} C_VEL
LIN {X 0,Y 160.781,Z 1165.31,A -85,B 0,C 180,E1 6819.889,E2 6819.889} C_VEL
LIN {X 0,Y 143.494,Z 1172.871,A -85,B 0,C 180,E1 6813.96,E2 6813.96} C_VEL
LIN {X 0,Y 128.082,Z 1179.167,A -85,B 0,C 180,E1 6806.645,E2 6806.645} C_VEL
LIN {X 0,Y 112.46,Z 1185.363,A -85,B 0,C 180,E1 6795.338,E2 6795.338} C_VEL
LIN {X 0,Y 101.987,Z 1189.478,A -85,B 0,C 180,E1 6781.965,E2 6781.965} C_VEL
LIN {X 0,Y 97.411,Z 1191.702,A -85,B 0,C 180,E1 6769.799,E2 6769.799} C_VEL
LIN {X 0,Y 96.099,Z 1192.825,A -85,B 0,C 180,E1 6758.376,E2 6758.376} C_VEL
LIN {X 0,Y 96.095,Z 1193.167,A -85,B 0,C 180,E1 6750,E2 6750} C_VEL
LIN {X 0,Y 96.105,Z 1192.804,A -85,B 0,C 180,E1 6741.264,E2 6741.264} C_VEL
LIN {X 0,Y 97.698,Z 1191.536,A -85,B 0,C 180,E1 6729.011,E2 6729.011} C_VEL
LIN {X 0,Y 104.67,Z 1188.38,A -85,B 0,C 180,E1 6713.683,E2 6713.683} C_VEL
LIN {X 0,Y 116.086,Z 1183.809,A -85,B 0,C 180,E1 6701.467,E2 6701.467} C_VEL
LIN {X 0,Y 129.396,Z 1178.58,A -85,B 0,C 180,E1 6692.621,E2 6692.621} C_VEL
LIN {X 0,Y 144.279,Z 1172.469,A -85,B 0,C 180,E1 6685.723,E2 6685.723} C_VEL
LIN {X 0,Y 163.246,Z 1164.13,A -85,B 0,C 180,E1 6679.4,E2 6679.4} C_VEL
LIN {X 0,Y 186.365,Z 1152.767,A -85,B 0,C 180,E1 6673.816,E2 6673.816} C_VEL
LIN {X 0,Y 205.306,Z 1142.442,A -85,B 0,C 180,E1 6670.341,E2 6670.341} C_VEL
LIN {X 0,Y 222.979,Z 1131.904,A -85,B 0,C 180,E1 6667.701,E2 6667.701} C_VEL
LIN {X 0,Y 242.017,Z 1119.48,A -85,B 0,C 180,E1 6665.344,E2 6665.344} C_VEL
LIN {X 0,Y 264.619,Z 1103.135,A -85,B 0,C 180,E1 6663.032,E2 6663.032} C_VEL
LIN {X 0,Y 285.031,Z 1086.461,A -85,B 0,C 180,E1 6661.291,E2 6661.291} C_VEL
LIN {X 0,Y 301.444,Z 1071.734,A -85,B 0,C 180,E1 6660.086,E2 6660.086} C_VEL
LIN {X 0,Y 311.378,Z 1062.208,A -85,B 0,C 180,E1 6659.419,E2 6659.419} C_VEL
LIN {X 0,Y 289.812,Z 1081.958,A -85,B 0,C 180,E1 6657.825,E2 6657.825} C_VEL
LIN {X 0,Y 272.513,Z 1096.155,A -85,B 0,C 180,E1 6656.351,E2 6656.351} C_VEL
LIN {X 0,Y 256.036,Z 1108.504,A -85,B 0,C 180,E1 6654.754,E2 6654.754} C_VEL
LIN {X 0,Y 238.27,Z 1120.659,A -85,B 0,C 180,E1 6652.768,E2 6652.768} C_VEL
LIN {X 0,Y 217.298,Z 1133.678,A -85,B 0,C 180,E1 6649.958,E2 6649.958} C_VEL
LIN {X 0,Y 194.624,Z 1146.094,A -85,B 0,C 180,E1 6646.159,E2 6646.159} C_VEL
LIN {X 0,Y 176.348,Z 1155.069,A -85,B 0,C 180,E1 6642.274,E2 6642.274} C_VEL
LIN {X 0,Y 159,Z 1162.816,A -85,B 0,C 180,E1 6637.577,E2 6637.577} C_VEL
LIN {X 0,Y 142.168,Z 1169.69,A -85,B 0,C 180,E1 6631.535,E2 6631.535} C_VEL
LIN {X 0,Y 123.421,Z 1176.703,A -85,B 0,C 180,E1 6621.796,E2 6621.796} C_VEL
LIN {X 0,Y 110.599,Z 1181.118,A -85,B 0,C 180,E1 6611.296,E2 6611.296} C_VEL
LIN {X 0,Y 102.234,Z 1184.038,A -85,B 0,C 180,E1 6599.92,E2 6599.92} C_VEL
LIN {X 0,Y 97.962,Z 1185.703,A -85,B 0,C 180,E1 6589.063,E2 6589.063} C_VEL
LIN {X 0,Y 96.322,Z 1186.57,A -85,B 0,C 180,E1 6578.356,E2 6578.356} C_VEL
LIN {X 0,Y 96.096,Z 1186.825,A -85,B 0,C 180,E1 6568.808,E2 6568.808} C_VEL
LIN {X 0,Y 96.583,Z 1186.485,A -85,B 0,C 180,E1 6558.656,E2 6558.656} C_VEL
LIN {X 0,Y 100.072,Z 1184.93,A -85,B 0,C 180,E1 6544.556,E2 6544.556} C_VEL
LIN {X 0,Y 107.919,Z 1182.083,A -85,B 0,C 180,E1 6531.629,E2 6531.629} C_VEL
LIN {X 0,Y 118.704,Z 1178.352,A -85,B 0,C 180,E1 6521.439,E2 6521.439} C_VEL
LIN {X 0,Y 131.617,Z 1173.734,A -85,B 0,C 180,E1 6513.318,E2 6513.318} C_VEL
LIN {X 0,Y 147.277,Z 1167.748,A -85,B 0,C 180,E1 6506.345,E2 6506.345} C_VEL
LIN {X 0,Y 167.89,Z 1159.147,A -85,B 0,C 180,E1 6499.787,E2 6499.787} C_VEL
LIN {X 0,Y 189.252,Z 1148.927,A -85,B 0,C 180,E1 6494.8,E2 6494.8} C_VEL
LIN {X 0,Y 207.156,Z 1139.495,A -85,B 0,C 180,E1 6491.538,E2 6491.538} C_VEL
LIN {X 0,Y 225.608,Z 1128.802,A -85,B 0,C 180,E1 6488.775,E2 6488.775} C_VEL
LIN {X 0,Y 247.364,Z 1114.878,A -85,B 0,C 180,E1 6486.098,E2 6486.098} C_VEL
LIN {X 0,Y 268.592,Z 1099.428,A -85,B 0,C 180,E1 6483.927,E2 6483.927} C_VEL
LIN {X 0,Y 286.206,Z 1085.252,A -85,B 0,C 180,E1 6482.385,E2 6482.385} C_VEL
LIN {X 0,Y 303.011,Z 1070.39,A -85,B 0,C 180,E1 6481.094,E2 6481.094} C_VEL
LIN {X 0,Y 310.756,Z 1063.13,A -85,B 0,C 180,E1 6480.53,E2 6480.53} C_VEL
LIN {X 0,Y 300.78,Z 1072.617,A -85,B 0,C 180,E1 6479.859,E2 6479.859} C_VEL
LIN {X 0,Y 295.106,Z 1077.92,A -85,B 0,C 180,E1 6479.658,E2 6479.658} C_VEL
LIN {X 0,Y 278.914,Z 1091.62,A -85,B 0,C 180,E1 6479.77,E2 6479.77} C_VEL
LIN {X 0,Y 273.782,Z 1095.62,A -85,B 0,C 180,E1 6479.541,E2 6479.541} C_VEL
LIN {X 0,Y 256.11,Z 1109.056,A -85,B 0,C 180,E1 6478.055,E2 6478.055} C_VEL
LIN {X 0,Y 238.454,Z 1121.31,A -85,B 0,C 180,E1 6476.331,E2 6476.331} C_VEL
LIN {X 0,Y 219.135,Z 1133.526,A -85,B 0,C 180,E1 6474.086,E2 6474.086} C_VEL
LIN {X 0,Y 195.565,Z 1146.953,A -85,B 0,C 180,E1 6470.659,E2 6470.659} C_VEL
LIN {X 0,Y 173.741,Z 1157.868,A -85,B 0,C 180,E1 6466.549,E2 6466.549} C_VEL
LIN {X 0,Y 155.269,Z 1166.242,A -85,B 0,C 180,E1 6461.994,E2 6461.994} C_VEL
LIN {X 0,Y 137.692,Z 1173.521,A -85,B 0,C 180,E1 6456.199,E2 6456.199} C_VEL
LIN {X 0,Y 118.221,Z 1180.975,A -85,B 0,C 180,E1 6446.855,E2 6446.855} C_VEL
LIN {X 0,Y 103.087,Z 1186.281,A -85,B 0,C 180,E1 6435.075,E2 6435.075} C_VEL
LIN {X 0,Y 94.387,Z 1189.452,A -85,B 0,C 180,E1 6423.425,E2 6423.425} C_VEL
LIN {X 0,Y 89.593,Z 1191.508,A -85,B 0,C 180,E1 6410.923,E2 6410.923} C_VEL
LIN {X 0,Y 88.118,Z 1192.56,A -85,B 0,C 180,E1 6399.14,E2 6399.14} C_VEL
LIN {X 0,Y 88.099,Z 1192.905,A -85,B 0,C 180,E1 6390,E2 6390} C_VEL
LIN {X 0,Y 88.118,Z 1192.554,A -85,B 0,C 180,E1 6380.826,E2 6380.826} C_VEL
LIN {X 0,Y 89.75,Z 1191.418,A -85,B 0,C 180,E1 6368.43,E2 6368.43} C_VEL
LIN {X 0,Y 95.776,Z 1188.936,A -85,B 0,C 180,E1 6354.224,E2 6354.224} C_VEL
LIN {X 0,Y 109.545,Z 1183.966,A -85,B 0,C 180,E1 6339.12,E2 6339.12} C_VEL
LIN {X 0,Y 124.352,Z 1178.568,A -85,B 0,C 180,E1 6329.73,E2 6329.73} C_VEL
LIN {X 0,Y 140.03,Z 1172.505,A -85,B 0,C 180,E1 6322.913,E2 6322.913} C_VEL
LIN {X 0,Y 158.073,Z 1164.946,A -85,B 0,C 180,E1 6317.231,E2 6317.231} C_VEL
LIN {X 0,Y 181.808,Z 1153.9,A -85,B 0,C 180,E1 6311.787,E2 6311.787} C_VEL
LIN {X 0,Y 203.02,Z 1142.69,A -85,B 0,C 180,E1 6308.147,E2 6308.147} C_VEL
LIN {X 0,Y 222.006,Z 1131.626,A -85,B 0,C 180,E1 6305.543,E2 6305.543} C_VEL
LIN {X 0,Y 241.701,Z 1118.988,A -85,B 0,C 180,E1 6303.32,E2 6303.32} C_VEL
LIN {X 0,Y 265.015,Z 1102.299,A -85,B 0,C 180,E1 6301.157,E2 6301.157} C_VEL
LIN {X 0,Y 285.138,Z 1086.036,A -85,B 0,C 180,E1 6299.598,E2 6299.598} C_VEL
LIN {X 0,Y 288.405,Z 1083.244,A -85,B 0,C 180,E1 6299.367,E2 6299.367} C_VEL
LIN {X 0,Y 271.125,Z 1097.187,A -85,B 0,C 180,E1 6298.005,E2 6298.005} C_VEL
LIN {X 0,Y 253.458,Z 1110.156,A -85,B 0,C 180,E1 6296.418,E2 6296.418} C_VEL
LIN {X 0,Y 233.13,Z 1123.681,A -85,B 0,C 180,E1 6294.272,E2 6294.272} C_VEL
LIN {X 0,Y 209.429,Z 1137.595,A -85,B 0,C 180,E1 6291.211,E2 6291.211} C_VEL
LIN {X 0,Y 190.068,Z 1147.711,A -85,B 0,C 180,E1 6288.085,E2 6288.085} C_VEL
LIN {X 0,Y 172.237,Z 1156.132,A -85,B 0,C 180,E1 6284.504,E2 6284.504} C_VEL
LIN {X 0,Y 153.524,Z 1164.118,A -85,B 0,C 180,E1 6279.69,E2 6279.69} C_VEL
LIN {X 0,Y 131.632,Z 1172.454,A -85,B 0,C 180,E1 6271.777,E2 6271.777} C_VEL
LIN {X 0,Y 115.281,Z 1177.961,A -85,B 0,C 180,E1 6262.933,E2 6262.933} C_VEL
LIN {X 0,Y 103.538,Z 1181.692,A -85,B 0,C 180,E1 6253.286,E2 6253.286} C_VEL
LIN {X 0,Y 94.881,Z 1184.413,A -85,B 0,C 180,E1 6241.796,E2 6241.796} C_VEL
LIN {X 0,Y 90.143,Z 1186.032,A -85,B 0,C 180,E1 6230.112,E2 6230.112} C_VEL
LIN {X 0,Y 88.374,Z 1186.834,A -85,B 0,C 180,E1 6219.114,E2 6219.114} C_VEL
LIN {X 0,Y 88.1,Z 1187.11,A -85,B 0,C 180,E1 6209.35,E2 6209.35} C_VEL
LIN {X 0,Y 88.538,Z 1186.786,A -85,B 0,C 180,E1 6198.932,E2 6198.932} C_VEL
LIN {X 0,Y 92.236,Z 1185.411,A -85,B 0,C 180,E1 6183.612,E2 6183.612} C_VEL
LIN {X 0,Y 101.58,Z 1182.353,A -85,B 0,C 180,E1 6168.74,E2 6168.74} C_VEL
LIN {X 0,Y 113.379,Z 1178.624,A -85,B 0,C 180,E1 6158.292,E2 6158.292} C_VEL
LIN {X 0,Y 127.233,Z 1174.006,A -85,B 0,C 180,E1 6150.182,E2 6150.182} C_VEL
LIN {X 0,Y 143.846,Z 1167.994,A -85,B 0,C 180,E1 6143.342,E2 6143.342} C_VEL
LIN {X 0,Y 166.106,Z 1159.026,A -85,B 0,C 180,E1 6136.847,E2 6136.847} C_VEL
LIN {X 0,Y 187.332,Z 1149.182,A -85,B 0,C 180,E1 6132.328,E2 6132.328} C_VEL
LIN {X 0,Y 205.942,Z 1139.61,A -85,B 0,C 180,E1 6129.22,E2 6129.22} C_VEL
LIN {X 0,Y 224.782,Z 1128.901,A -85,B 0,C 180,E1 6126.641,E2 6126.641} C_VEL
LIN {X 0,Y 247.593,Z 1114.502,A -85,B 0,C 180,E1 6124.084,E2 6124.084} C_VEL
LIN {X 0,Y 269.138,Z 1098.938,A -85,B 0,C 180,E1 6122.081,E2 6122.081} C_VEL
LIN {X 0,Y 285.982,Z 1085.52,A -85,B 0,C 180,E1 6120.733,E2 6120.733} C_VEL
LIN {X 0,Y 287.748,Z 1084.045,A -85,B 0,C 180,E1 6120.578,E2 6120.578} C_VEL
LIN {X 0,Y 273.782,Z 1095.62,A -85,B 0,C 180,E1 6119.541,E2 6119.541} C_VEL
LIN {X 0,Y 267.715,Z 1100.349,A -85,B 0,C 180,E1 6119.282,E2 6119.282} C_VEL
LIN {X 0,Y 250.536,Z 1112.812,A -85,B 0,C 180,E1 6119.294,E2 6119.294} C_VEL
LIN {X 0,Y 245.107,Z 1116.441,A -85,B 0,C 180,E1 6119.003,E2 6119.003} C_VEL
LIN {X 0,Y 223.307,Z 1130.325,A -85,B 0,C 180,E1 6116.838,E2 6116.838} C_VEL
LIN {X 0,Y 203.917,Z 1141.487,A -85,B 0,C 180,E1 6114.478,E2 6114.478} C_VEL
LIN {X 0,Y 184.003,Z 1151.854,A -85,B 0,C 180,E1 6111.483,E2 6111.483} C_VEL
LIN {X 0,Y 160.215,Z 1162.934,A -85,B 0,C 180,E1 6106.793,E2 6106.793} C_VEL
LIN {X 0,Y 138.624,Z 1171.674,A -85,B 0,C 180,E1 6100.885,E2 6100.885} C_VEL
LIN {X 0,Y 121.901,Z 1177.82,A -85,B 0,C 180,E1 6094.454,E2 6094.454} C_VEL
LIN {X 0,Y 107.026,Z 1182.871,A -85,B 0,C 180,E1 6086.248,E2 6086.248} C_VEL
LIN {X 0,Y 94.209,Z 1187.024,A -85,B 0,C 180,E1 6075.323,E2 6075.323} C_VEL
LIN {X 0,Y 84.306,Z 1190.402,A -85,B 0,C 180,E1 6059.875,E2 6059.875} C_VEL
LIN {X 0,Y 80.376,Z 1192.155,A -85,B 0,C 180,E1 6043.671,E2 6043.671} C_VEL
LIN {X 0,Y 80.079,Z 1192.563,A -85,B 0,C 180,E1 6032.67,E2 6032.67} C_VEL
LIN {X 0,Y 80.064,Z 1192.476,A -85,B 0,C 180,E1 6024.985,E2 6024.985} C_VEL
LIN {X 0,Y 80.809,Z 1191.823,A -85,B 0,C 180,E1 6012.725,E2 6012.725} C_VEL
LIN {X 0,Y 85.612,Z 1189.846,A -85,B 0,C 180,E1 5997.236,E2 5997.236} C_VEL
LIN {X 0,Y 94.715,Z 1186.817,A -85,B 0,C 180,E1 5984.124,E2 5984.124} C_VEL
LIN {X 0,Y 107.024,Z 1182.823,A -85,B 0,C 180,E1 5973.75,E2 5973.75} C_VEL
LIN {X 0,Y 121.897,Z 1177.759,A -85,B 0,C 180,E1 5965.542,E2 5965.542} C_VEL
LIN {X 0,Y 139.573,Z 1171.24,A -85,B 0,C 180,E1 5958.807,E2 5958.807} C_VEL
LIN {X 0,Y 162.895,Z 1161.655,A -85,B 0,C 180,E1 5952.592,E2 5952.592} C_VEL
LIN {X 0,Y 184.937,Z 1151.269,A -85,B 0,C 180,E1 5948.356,E2 5948.356} C_VEL
LIN {X 0,Y 203.915,Z 1141.358,A -85,B 0,C 180,E1 5945.516,E2 5945.516} C_VEL
LIN {X 0,Y 223.306,Z 1130.177,A -85,B 0,C 180,E1 5943.155,E2 5943.155} C_VEL
LIN {X 0,Y 246.99,Z 1115.001,A -85,B 0,C 180,E1 5940.823,E2 5940.823} C_VEL
LIN {X 0,Y 265.347,Z 1101.735,A -85,B 0,C 180,E1 5939.318,E2 5939.318} C_VEL
LIN {X 0,Y 242.234,Z 1117.723,A -85,B 0,C 180,E1 5937.3,E2 5937.3} C_VEL
LIN {X 0,Y 222.732,Z 1129.734,A -85,B 0,C 180,E1 5935.251,E2 5935.251} C_VEL
LIN {X 0,Y 204.51,Z 1139.884,A -85,B 0,C 180,E1 5932.965,E2 5932.965} C_VEL
LIN {X 0,Y 185.531,Z 1149.428,A -85,B 0,C 180,E1 5930.069,E2 5930.069} C_VEL
LIN {X 0,Y 162.161,Z 1159.94,A -85,B 0,C 180,E1 5925.473,E2 5925.473} C_VEL
LIN {X 0,Y 139.909,Z 1168.483,A -85,B 0,C 180,E1 5919.421,E2 5919.421} C_VEL
LIN {X 0,Y 122.786,Z 1174.366,A -85,B 0,C 180,E1 5912.869,E2 5912.869} C_VEL
LIN {X 0,Y 107.84,Z 1179.021,A -85,B 0,C 180,E1 5904.677,E2 5904.677} C_VEL
LIN {X 0,Y 94.572,Z 1182.869,A -85,B 0,C 180,E1 5893.41,E2 5893.41} C_VEL
LIN {X 0,Y 84.188,Z 1185.868,A -85,B 0,C 180,E1 5876.827,E2 5876.827} C_VEL
LIN {X 0,Y 80.561,Z 1187.064,A -85,B 0,C 180,E1 5861.327,E2 5861.327} C_VEL
LIN {X 0,Y 80.11,Z 1187.383,A -85,B 0,C 180,E1 5850,E2 5850} C_VEL
LIN {X 0,Y 80.564,Z 1187.069,A -85,B 0,C 180,E1 5838.547,E2 5838.547} C_VEL
LIN {X 0,Y 84.427,Z 1185.832,A -85,B 0,C 180,E1 5822.492,E2 5822.492} C_VEL
LIN {X 0,Y 95.022,Z 1182.774,A -85,B 0,C 180,E1 5806.015,E2 5806.015} C_VEL
LIN {X 0,Y 107.779,Z 1179.093,A -85,B 0,C 180,E1 5795.277,E2 5795.277} C_VEL
LIN {X 0,Y 123.254,Z 1174.279,A -85,B 0,C 180,E1 5786.832,E2 5786.832} C_VEL
LIN {X 0,Y 140.675,Z 1168.294,A -85,B 0,C 180,E1 5780.249,E2 5780.249} C_VEL
LIN {X 0,Y 163.881,Z 1159.298,A -85,B 0,C 180,E1 5774.053,E2 5774.053} C_VEL
LIN {X 0,Y 185.694,Z 1149.472,A -85,B 0,C 180,E1 5769.821,E2 5769.821} C_VEL
LIN {X 0,Y 204.477,Z 1140.039,A -85,B 0,C 180,E1 5766.959,E2 5766.959} C_VEL
LIN {X 0,Y 223.676,Z 1129.344,A -85,B 0,C 180,E1 5764.562,E2 5764.562} C_VEL
LIN {X 0,Y 246.155,Z 1115.418,A -85,B 0,C 180,E1 5762.257,E2 5762.257} C_VEL
LIN {X 0,Y 264.835,Z 1102.352,A -85,B 0,C 180,E1 5760.635,E2 5760.635} C_VEL
LIN {X 0,Y 245.107,Z 1116.441,A -85,B 0,C 180,E1 5759.003,E2 5759.003} C_VEL
LIN {X 0,Y 238.659,Z 1120.643,A -85,B 0,C 180,E1 5758.669,E2 5758.669} C_VEL
LIN {X 0,Y 221.436,Z 1131.063,A -85,B 0,C 180,E1 5758.577,E2 5758.577} C_VEL
LIN {X 0,Y 214.901,Z 1134.835,A -85,B 0,C 180,E1 5758.166,E2 5758.166} C_VEL
LIN {X 0,Y 189.673,Z 1148.284,A -85,B 0,C 180,E1 5755.075,E2 5755.075} C_VEL
LIN {X 0,Y 169.289,Z 1157.897,A -85,B 0,C 180,E1 5751.851,E2 5751.851} C_VEL
LIN {X 0,Y 150.283,Z 1165.94,A -85,B 0,C 180,E1 5747.963,E2 5747.963} C_VEL
LIN {X 0,Y 130.08,Z 1173.597,A -85,B 0,C 180,E1 5742.386,E2 5742.386} C_VEL
LIN {X 0,Y 106.936,Z 1181.293,A -85,B 0,C 180,E1 5732.654,E2 5732.654} C_VEL
LIN {X 0,Y 91.452,Z 1185.903,A -85,B 0,C 180,E1 5721.923,E2 5721.923} C_VEL
LIN {X 0,Y 80.651,Z 1189.031,A -85,B 0,C 180,E1 5709.217,E2 5709.217} C_VEL
LIN {X 0,Y 74.294,Z 1191.046,A -85,B 0,C 180,E1 5694.658,E2 5694.658} C_VEL
LIN {X 0,Y 72.159,Z 1192.06,A -85,B 0,C 180,E1 5680.316,E2 5680.316} C_VEL
LIN {X 0,Y 72.106,Z 1192.38,A -85,B 0,C 180,E1 5670,E2 5670} C_VEL
LIN {X 0,Y 72.161,Z 1192.052,A -85,B 0,C 180,E1 5659.623,E2 5659.623} C_VEL
LIN {X 0,Y 74.294,Z 1191.03,A -85,B 0,C 180,E1 5645.342,E2 5645.342} C_VEL
LIN {X 0,Y 80.651,Z 1189.004,A -85,B 0,C 180,E1 5630.783,E2 5630.783} C_VEL
LIN {X 0,Y 92.055,Z 1185.695,A -85,B 0,C 180,E1 5617.543,E2 5617.543} C_VEL
LIN {X 0,Y 110.686,Z 1180.135,A -85,B 0,C 180,E1 5605.402,E2 5605.402} C_VEL
LIN {X 0,Y 131.782,Z 1172.892,A -85,B 0,C 180,E1 5597.062,E2 5597.062} C_VEL
LIN {X 0,Y 150.281,Z 1165.848,A -85,B 0,C 180,E1 5592.033,E2 5592.033} C_VEL
LIN {X 0,Y 169.659,Z 1157.626,A -85,B 0,C 180,E1 5588.078,E2 5588.078} C_VEL
LIN {X 0,Y 191.603,Z 1147.226,A -85,B 0,C 180,E1 5584.65,E2 5584.65} C_VEL
LIN {X 0,Y 217.181,Z 1133.334,A -85,B 0,C 180,E1 5581.583,E2 5581.583} C_VEL
LIN {X 0,Y 236.969,Z 1121.234,A -85,B 0,C 180,E1 5579.7,E2 5579.7} C_VEL
LIN {X 0,Y 241.985,Z 1117.997,A -85,B 0,C 180,E1 5579.261,E2 5579.261} C_VEL
LIN {X 0,Y 222.199,Z 1130.009,A -85,B 0,C 180,E1 5577.387,E2 5577.387} C_VEL
LIN {X 0,Y 203.658,Z 1140.158,A -85,B 0,C 180,E1 5575.29,E2 5575.29} C_VEL
LIN {X 0,Y 184.488,Z 1149.603,A -85,B 0,C 180,E1 5572.654,E2 5572.654} C_VEL
LIN {X 0,Y 161.185,Z 1159.833,A -85,B 0,C 180,E1 5568.55,E2 5568.55} C_VEL
LIN {X 0,Y 138.06,Z 1168.466,A -85,B 0,C 180,E1 5562.934,E2 5562.934} C_VEL
LIN {X 0,Y 119.781,Z 1174.467,A -85,B 0,C 180,E1 5556.665,E2 5556.665} C_VEL
LIN {X 0,Y 103.262,Z 1179.295,A -85,B 0,C 180,E1 5548.439,E2 5548.439} C_VEL
LIN {X 0,Y 88.211,Z 1183.291,A -85,B 0,C 180,E1 5536.505,E2 5536.505} C_VEL
LIN {X 0,Y 76.392,Z 1186.259,A -85,B 0,C 180,E1 5518.111,E2 5518.111} C_VEL
LIN {X 0,Y 72.604,Z 1187.344,A -85,B 0,C 180,E1 5501.921,E2 5501.921} C_VEL
LIN {X 0,Y 72.114,Z 1187.646,A -85,B 0,C 180,E1 5490,E2 5490} C_VEL
LIN {X 0,Y 72.617,Z 1187.347,A -85,B 0,C 180,E1 5477.858,E2 5477.858} C_VEL
LIN {X 0,Y 76.957,Z 1186.161,A -85,B 0,C 180,E1 5460.415,E2 5460.415} C_VEL
LIN {X 0,Y 88.71,Z 1183.196,A -85,B 0,C 180,E1 5442.893,E2 5442.893} C_VEL
LIN {X 0,Y 103.206,Z 1179.364,A -85,B 0,C 180,E1 5431.511,E2 5431.511} C_VEL
LIN {X 0,Y 119.725,Z 1174.552,A -85,B 0,C 180,E1 5423.272,E2 5423.272} C_VEL
LIN {X 0,Y 138.009,Z 1168.567,A -85,B 0,C 180,E1 5416.997,E2 5416.997} C_VEL
LIN {X 0,Y 162.057,Z 1159.571,A -85,B 0,C 180,E1 5411.19,E2 5411.19} C_VEL
LIN {X 0,Y 184.456,Z 1149.744,A -85,B 0,C 180,E1 5407.268,E2 5407.268} C_VEL
LIN {X 0,Y 203.635,Z 1140.31,A -85,B 0,C 180,E1 5404.632,E2 5404.632} C_VEL
LIN {X 0,Y 223.169,Z 1129.615,A -85,B 0,C 180,E1 5402.434,E2 5402.434} C_VEL
LIN {X 0,Y 241.568,Z 1118.443,A -85,B 0,C 180,E1 5400.681,E2 5400.681} C_VEL
LIN {X 0,Y 222.008,Z 1130.636,A -85,B 0,C 180,E1 5398.901,E2 5398.901} C_VEL
LIN {X 0,Y 214.901,Z 1134.835,A -85,B 0,C 180,E1 5398.166,E2 5398.166} C_VEL
LIN {X 0,Y 208.286,Z 1138.548,A -85,B 0,C 180,E1 5397.721,E2 5397.721} C_VEL
LIN {X 0,Y 190.274,Z 1147.529,A -85,B 0,C 180,E1 5397.443,E2 5397.443} C_VEL
LIN {X 0,Y 183.451,Z 1150.734,A -85,B 0,C 180,E1 5396.897,E2 5396.897} C_VEL
LIN {X 0,Y 159.05,Z 1161.651,A -85,B 0,C 180,E1 5393.14,E2 5393.14} C_VEL
LIN {X 0,Y 134.949,Z 1170.807,A -85,B 0,C 180,E1 5387.961,E2 5387.961} C_VEL
LIN {X 0,Y 115.634,Z 1177.268,A -85,B 0,C 180,E1 5382.015,E2 5382.015} C_VEL
LIN {X 0,Y 97.927,Z 1182.538,A -85,B 0,C 180,E1 5373.961,E2 5373.961} C_VEL
LIN {X 0,Y 81.48,Z 1186.986,A -85,B 0,C 180,E1 5361.753,E2 5361.753} C_VEL
LIN {X 0,Y 68.497,Z 1190.363,A -85,B 0,C 180,E1 5342.149,E2 5342.149} C_VEL
LIN {X 0,Y 64.332,Z 1191.736,A -85,B 0,C 180,E1 5323.481,E2 5323.481} C_VEL
LIN {X 0,Y 64.093,Z 1192.08,A -85,B 0,C 180,E1 5311.788,E2 5311.788} C_VEL
LIN {X 0,Y 64.105,Z 1191.896,A -85,B 0,C 180,E1 5301.93,E2 5301.93} C_VEL
LIN {X 0,Y 65.782,Z 1191.137,A -85,B 0,C 180,E1 5286.722,E2 5286.722} C_VEL
LIN {X 0,Y 72.549,Z 1189.221,A -85,B 0,C 180,E1 5269.629,E2 5269.629} C_VEL
LIN {X 0,Y 84.487,Z 1186.126,A -85,B 0,C 180,E1 5255.444,E2 5255.444} C_VEL
LIN {X 0,Y 99.449,Z 1182.053,A -85,B 0,C 180,E1 5245.197,E2 5245.197} C_VEL
LIN {X 0,Y 117.41,Z 1176.65,A -85,B 0,C 180,E1 5237.342,E2 5237.342} C_VEL
LIN {X 0,Y 141.332,Z 1168.486,A -85,B 0,C 180,E1 5230.469,E2 5230.469} C_VEL
LIN {X 0,Y 164.837,Z 1159.014,A -85,B 0,C 180,E1 5225.857,E2 5225.857} C_VEL
LIN {X 0,Y 185.205,Z 1149.77,A -85,B 0,C 180,E1 5222.867,E2 5222.867} C_VEL
LIN {X 0,Y 205.004,Z 1139.735,A -85,B 0,C 180,E1 5220.559,E2 5220.559} C_VEL
LIN {X 0,Y 218.569,Z 1132.205,A -85,B 0,C 180,E1 5219.214,E2 5219.214} C_VEL
LIN {X 0,Y 194.312,Z 1144.953,A -85,B 0,C 180,E1 5216.61,E2 5216.61} C_VEL
LIN {X 0,Y 170.026,Z 1155.828,A -85,B 0,C 180,E1 5213.245,E2 5213.245} C_VEL
LIN {X 0,Y 150.309,Z 1163.612,A -85,B 0,C 180,E1 5209.653,E2 5209.653} C_VEL
LIN {X 0,Y 130.786,Z 1170.405,A -85,B 0,C 180,E1 5204.934,E2 5204.934} C_VEL
LIN {X 0,Y 108.525,Z 1177.182,A -85,B 0,C 180,E1 5197.118,E2 5197.118} C_VEL
LIN {X 0,Y 88.492,Z 1182.205,A -85,B 0,C 180,E1 5185.57,E2 5185.57} C_VEL
LIN {X 0,Y 75.57,Z 1185.117,A -85,B 0,C 180,E1 5172.437,E2 5172.437} C_VEL
LIN {X 0,Y 67.744,Z 1186.833,A -85,B 0,C 180,E1 5157.228,E2 5157.228} C_VEL
LIN {X 0,Y 64.55,Z 1187.646,A -85,B 0,C 180,E1 5141.617,E2 5141.617} C_VEL
LIN {X 0,Y 64.112,Z 1187.897,A -85,B 0,C 180,E1 5129.106,E2 5129.106} C_VEL
LIN {X 0,Y 64.83,Z 1187.599,A -85,B 0,C 180,E1 5115.714,E2 5115.714} C_VEL
LIN {X 0,Y 70.707,Z 1186.306,A -85,B 0,C 180,E1 5095.554,E2 5095.554} C_VEL
LIN {X 0,Y 83.923,Z 1183.315,A -85,B 0,C 180,E1 5078.157,E2 5078.157} C_VEL
LIN {X 0,Y 99.119,Z 1179.636,A -85,B 0,C 180,E1 5067.416,E2 5067.416} C_VEL
LIN {X 0,Y 116.685,Z 1174.824,A -85,B 0,C 180,E1 5059.512,E2 5059.512} C_VEL
LIN {X 0,Y 135.801,Z 1168.84,A -85,B 0,C 180,E1 5053.623,E2 5053.623} C_VEL
LIN {X 0,Y 160.648,Z 1159.844,A -85,B 0,C 180,E1 5048.271,E2 5048.271} C_VEL
LIN {X 0,Y 183.586,Z 1150.016,A -85,B 0,C 180,E1 5044.684,E2 5044.684} C_VEL
LIN {X 0,Y 203.441,Z 1140.425,A -85,B 0,C 180,E1 5042.253,E2 5042.253} C_VEL
LIN {X 0,Y 218.236,Z 1132.555,A -85,B 0,C 180,E1 5040.737,E2 5040.737} C_VEL
LIN {X 0,Y 193.077,Z 1146.125,A -85,B 0,C 180,E1 5038.109,E2 5038.109} C_VEL
LIN {X 0,Y 183.451,Z 1150.734,A -85,B 0,C 180,E1 5036.897,E2 5036.897} C_VEL
LIN {X 0,Y 176.599,Z 1153.967,A -85,B 0,C 180,E1 5036.304,E2 5036.304} C_VEL
LIN {X 0,Y 156.986,Z 1161.924,A -85,B 0,C 180,E1 5035.685,E2 5035.685} C_VEL
LIN {X 0,Y 151.011,Z 1164.126,A -85,B 0,C 180,E1 5034.99,E2 5034.99} C_VEL
LIN {X 0,Y 130.638,Z 1171.473,A -85,B 0,C 180,E1 5030.865,E2 5030.865} C_VEL
LIN {X 0,Y 110.66,Z 1177.788,A -85,B 0,C 180,E1 5025.192,E2 5025.192} C_VEL
LIN {X 0,Y 88.196,Z 1183.991,A -85,B 0,C 180,E1 5015.086,E2 5015.086} C_VEL
LIN {X 0,Y 69.725,Z 1188.241,A -85,B 0,C 180,E1 4999.466,E2 4999.466} C_VEL
LIN {X 0,Y 60.08,Z 1190.432,A -85,B 0,C 180,E1 4982.178,E2 4982.178} C_VEL
LIN {X 0,Y 56.383,Z 1191.498,A -85,B 0,C 180,E1 4964.375,E2 4964.375} C_VEL
LIN {X 0,Y 56.102,Z 1191.841,A -85,B 0,C 180,E1 4951.021,E2 4951.021} C_VEL
LIN {X 0,Y 56.194,Z 1191.576,A -85,B 0,C 180,E1 4938.713,E2 4938.713} C_VEL
LIN {X 0,Y 58.879,Z 1190.718,A -85,B 0,C 180,E1 4921.609,E2 4921.609} C_VEL
LIN {X 0,Y 66.976,Z 1188.826,A -85,B 0,C 180,E1 4904.228,E2 4904.228} C_VEL
LIN {X 0,Y 80.044,Z 1185.824,A -85,B 0,C 180,E1 4890.47,E2 4890.47} C_VEL
LIN {X 0,Y 96.17,Z 1181.776,A -85,B 0,C 180,E1 4880.658,E2 4880.658} C_VEL
LIN {X 0,Y 115.098,Z 1176.396,A -85,B 0,C 180,E1 4873.359,E2 4873.359} C_VEL
LIN {X 0,Y 140.044,Z 1168.208,A -85,B 0,C 180,E1 4867.067,E2 4867.067} C_VEL
LIN {X 0,Y 164.189,Z 1158.735,A -85,B 0,C 180,E1 4862.917,E2 4862.917} C_VEL
LIN {X 0,Y 184.975,Z 1149.491,A -85,B 0,C 180,E1 4860.249,E2 4860.249} C_VEL
LIN {X 0,Y 194.992,Z 1144.735,A -85,B 0,C 180,E1 4859.172,E2 4859.172} C_VEL
LIN {X 0,Y 170.349,Z 1155.659,A -85,B 0,C 180,E1 4856.205,E2 4856.205} C_VEL
LIN {X 0,Y 150.095,Z 1163.507,A -85,B 0,C 180,E1 4853.008,E2 4853.008} C_VEL
LIN {X 0,Y 130.422,Z 1170.185,A -85,B 0,C 180,E1 4848.898,E2 4848.898} C_VEL
LIN {X 0,Y 110.717,Z 1175.992,A -85,B 0,C 180,E1 4843.187,E2 4843.187} C_VEL
LIN {X 0,Y 88.569,Z 1181.575,A -85,B 0,C 180,E1 4833.104,E2 4833.104} C_VEL
LIN {X 0,Y 70.867,Z 1185.176,A -85,B 0,C 180,E1 4818.397,E2 4818.397} C_VEL
LIN {X 0,Y 60.957,Z 1187.04,A -85,B 0,C 180,E1 4801.66,E2 4801.66} C_VEL
LIN {X 0,Y 56.685,Z 1187.91,A -85,B 0,C 180,E1 4783.256,E2 4783.256} C_VEL
LIN {X 0,Y 56.116,Z 1188.159,A -85,B 0,C 180,E1 4768.979,E2 4768.979} C_VEL
LIN {X 0,Y 57.033,Z 1187.864,A -85,B 0,C 180,E1 4753.71,E2 4753.71} C_VEL
LIN {X 0,Y 64.12,Z 1186.574,A -85,B 0,C 180,E1 4731.411,E2 4731.411} C_VEL
LIN {X 0,Y 79.777,Z 1183.435,A -85,B 0,C 180,E1 4712.889,E2 4712.889} C_VEL
LIN {X 0,Y 96.509,Z 1179.682,A -85,B 0,C 180,E1 4702.541,E2 4702.541} C_VEL
LIN {X 0,Y 115.055,Z 1174.853,A -85,B 0,C 180,E1 4695.288,E2 4695.288} C_VEL
LIN {X 0,Y 137.802,Z 1167.943,A -85,B 0,C 180,E1 4689.328,E2 4689.328} C_VEL
LIN {X 0,Y 163.527,Z 1158.54,A -85,B 0,C 180,E1 4684.703,E2 4684.703} C_VEL
LIN {X 0,Y 184.081,Z 1149.841,A -85,B 0,C 180,E1 4681.96,E2 4681.96} C_VEL
LIN {X 0,Y 194.621,Z 1145.065,A -85,B 0,C 180,E1 4680.783,E2 4680.783} C_VEL
LIN {X 0,Y 170.088,Z 1156.345,A -85,B 0,C 180,E1 4677.91,E2 4677.91} C_VEL
LIN {X 0,Y 151.011,Z 1164.126,A -85,B 0,C 180,E1 4674.99,E2 4674.99} C_VEL
LIN {X 0,Y 144.003,Z 1166.72,A -85,B 0,C 180,E1 4674.148,E2 4674.148} C_VEL
LIN {X 0,Y 123.947,Z 1173.173,A -85,B 0,C 180,E1 4672.978,E2 4672.978} C_VEL
LIN {X 0,Y 117.9,Z 1174.923,A -85,B 0,C 180,E1 4671.945,E2 4671.945} C_VEL
LIN {X 0,Y 95.288,Z 1181.118,A -85,B 0,C 180,E1 4664.873,E2 4664.873} C_VEL
LIN {X 0,Y 76.921,Z 1185.421,A -85,B 0,C 180,E1 4655.49,E2 4655.49} C_VEL
LIN {X 0,Y 61.473,Z 1188.583,A -85,B 0,C 180,E1 4641.326,E2 4641.326} C_VEL
LIN {X 0,Y 51.147,Z 1190.617,A -85,B 0,C 180,E1 4620.548,E2 4620.548} C_VEL
LIN {X 0,Y 48.114,Z 1191.426,A -85,B 0,C 180,E1 4598.364,E2 4598.364} C_VEL
LIN {X 0,Y 48.091,Z 1191.549,A -85,B 0,C 180,E1 4587.617,E2 4587.617} C_VEL
LIN {X 0,Y 48.82,Z 1191.168,A -85,B 0,C 180,E1 4570.872,E2 4570.872} C_VEL
LIN {X 0,Y 56.463,Z 1189.609,A -85,B 0,C 180,E1 4546.321,E2 4546.321} C_VEL
LIN {X 0,Y 73.845,Z 1186.058,A -85,B 0,C 180,E1 4526.666,E2 4526.666} C_VEL
LIN {X 0,Y 92.251,Z 1181.82,A -85,B 0,C 180,E1 4516.368,E2 4516.368} C_VEL
LIN {X 0,Y 111.585,Z 1176.649,A -85,B 0,C 180,E1 4509.717,E2 4509.717} C_VEL
LIN {X 0,Y 133.06,Z 1169.973,A -85,B 0,C 180,E1 4504.742,E2 4504.742} C_VEL
LIN {X 0,Y 160.98,Z 1159.706,A -85,B 0,C 180,E1 4500.347,E2 4500.347} C_VEL
LIN {X 0,Y 170.747,Z 1155.638,A -85,B 0,C 180,E1 4499.099,E2 4499.099} C_VEL
LIN {X 0,Y 149.083,Z 1163.861,A -85,B 0,C 180,E1 4496.154,E2 4496.154} C_VEL
LIN {X 0,Y 128.385,Z 1170.673,A -85,B 0,C 180,E1 4492.392,E2 4492.392} C_VEL
LIN {X 0,Y 106.79,Z 1176.754,A -85,B 0,C 180,E1 4486.839,E2 4486.839} C_VEL
LIN {X 0,Y 81.62,Z 1182.5,A -85,B 0,C 180,E1 4476.155,E2 4476.155} C_VEL
LIN {X 0,Y 65.037,Z 1185.552,A -85,B 0,C 180,E1 4463.076,E2 4463.076} C_VEL
LIN {X 0,Y 53.765,Z 1187.369,A -85,B 0,C 180,E1 4445.205,E2 4445.205} C_VEL
LIN {X 0,Y 48.87,Z 1188.175,A -85,B 0,C 180,E1 4425.425,E2 4425.425} C_VEL
LIN {X 0,Y 48.12,Z 1188.422,A -85,B 0,C 180,E1 4408.809,E2 4408.809} C_VEL
LIN {X 0,Y 49.323,Z 1188.129,A -85,B 0,C 180,E1 4391.074,E2 4391.074} C_VEL
LIN {X 0,Y 57.938,Z 1186.843,A -85,B 0,C 180,E1 4366.346,E2 4366.346} C_VEL
LIN {X 0,Y 75.607,Z 1183.706,A -85,B 0,C 180,E1 4347.621,E2 4347.621} C_VEL
LIN {X 0,Y 93.509,Z 1179.983,A -85,B 0,C 180,E1 4337.891,E2 4337.891} C_VEL
LIN {X 0,Y 113.143,Z 1175.125,A -85,B 0,C 180,E1 4331.211,E2 4331.211} C_VEL
LIN {X 0,Y 136.698,Z 1168.216,A -85,B 0,C 180,E1 4325.875,E2 4325.875} C_VEL
LIN {X 0,Y 163.203,Z 1158.754,A -85,B 0,C 180,E1 4321.755,E2 4321.755} C_VEL
LIN {X 0,Y 170.61,Z 1155.812,A -85,B 0,C 180,E1 4320.83,E2 4320.83} C_VEL
LIN {X 0,Y 149.071,Z 1164.381,A -85,B 0,C 180,E1 4317.984,E2 4317.984} C_VEL
LIN {X 0,Y 128.603,Z 1171.511,A -85,B 0,C 180,E1 4314.363,E2 4314.363} C_VEL
LIN {X 0,Y 117.9,Z 1174.923,A -85,B 0,C 180,E1 4311.945,E2 4311.945} C_VEL
LIN {X 0,Y 110.818,Z 1176.89,A -85,B 0,C 180,E1 4310.656,E2 4310.656} C_VEL
LIN {X 0,Y 90.505,Z 1181.634,A -85,B 0,C 180,E1 4308.309,E2 4308.309} C_VEL
LIN {X 0,Y 84.552,Z 1182.961,A -85,B 0,C 180,E1 4306.571,E2 4306.571} C_VEL
LIN {X 0,Y 61.746,Z 1187.449,A -85,B 0,C 180,E1 4292.952,E2 4292.952} C_VEL
LIN {X 0,Y 47.469,Z 1189.815,A -85,B 0,C 180,E1 4274.035,E2 4274.035} C_VEL
LIN {X 0,Y 40.838,Z 1190.964,A -85,B 0,C 180,E1 4250.046,E2 4250.046} C_VEL
LIN {X 0,Y 40.101,Z 1191.316,A -85,B 0,C 180,E1 4231.429,E2 4231.429} C_VEL
LIN {X 0,Y 40.25,Z 1191.1,A -85,B 0,C 180,E1 4217.081,E2 4217.081} C_VEL
LIN {X 0,Y 44.679,Z 1190.254,A -85,B 0,C 180,E1 4192.827,E2 4192.827} C_VEL
LIN {X 0,Y 56.908,Z 1188.235,A -85,B 0,C 180,E1 4171.81,E2 4171.81} C_VEL
LIN {X 0,Y 73.839,Z 1185.103,A -85,B 0,C 180,E1 4158.581,E2 4158.581} C_VEL
LIN {X 0,Y 93.445,Z 1180.788,A -85,B 0,C 180,E1 4150.136,E2 4150.136} C_VEL
LIN {X 0,Y 119.207,Z 1173.974,A -85,B 0,C 180,E1 4143.512,E2 4143.512} C_VEL
LIN {X 0,Y 144.99,Z 1165.462,A -85,B 0,C 180,E1 4139.285,E2 4139.285} C_VEL
LIN {X 0,Y 146.557,Z 1164.893,A -85,B 0,C 180,E1 4139.075,E2 4139.075} C_VEL
LIN {X 0,Y 124.362,Z 1171.905,A -85,B 0,C 180,E1 4135.521,E2 4135.521} C_VEL
LIN {X 0,Y 96.033,Z 1179.178,A -85,B 0,C 180,E1 4128.59,E2 4128.59} C_VEL
LIN {X 0,Y 75.512,Z 1183.324,A -85,B 0,C 180,E1 4120.07,E2 4120.07} C_VEL
LIN {X 0,Y 59.004,Z 1186.034,A -85,B 0,C 180,E1 4107.917,E2 4107.917} C_VEL
LIN {X 0,Y 46.797,Z 1187.704,A -85,B 0,C 180,E1 4089.717,E2 4089.717} C_VEL
LIN {X 0,Y 40.973,Z 1188.458,A -85,B 0,C 180,E1 4067.028,E2 4067.028} C_VEL
LIN {X 0,Y 40.124,Z 1188.684,A -85,B 0,C 180,E1 4048.572,E2 4048.572} C_VEL
LIN {X 0,Y 41.524,Z 1188.412,A -85,B 0,C 180,E1 4028.827,E2 4028.827} C_VEL
LIN {X 0,Y 51.106,Z 1187.234,A -85,B 0,C 180,E1 4001.975,E2 4001.975} C_VEL
LIN {X 0,Y 71.471,Z 1184.1,A -85,B 0,C 180,E1 3982.194,E2 3982.194} C_VEL
LIN {X 0,Y 91.297,Z 1180.256,A -85,B 0,C 180,E1 3972.917,E2 3972.917} C_VEL
LIN {X 0,Y 111.82,Z 1175.399,A -85,B 0,C 180,E1 3967.012,E2 3967.012} C_VEL
LIN {X 0,Y 135.112,Z 1168.782,A -85,B 0,C 180,E1 3962.533,E2 3962.533} C_VEL
LIN {X 0,Y 146.274,Z 1165.097,A -85,B 0,C 180,E1 3960.881,E2 3960.881} C_VEL
LIN {X 0,Y 122.144,Z 1173.121,A -85,B 0,C 180,E1 3957.055,E2 3957.055} C_VEL
LIN {X 0,Y 95.303,Z 1180.408,A -85,B 0,C 180,E1 3950.465,E2 3950.465} C_VEL
LIN {X 0,Y 84.552,Z 1182.961,A -85,B 0,C 180,E1 3946.571,E2 3946.571} C_VEL
LIN {X 0,Y 77.631,Z 1184.407,A -85,B 0,C 180,E1 3944.306,E2 3944.306} C_VEL
LIN {X 0,Y 57.099,Z 1187.44,A -85,B 0,C 180,E1 3938.464,E2 3938.464} C_VEL
LIN {X 0,Y 52.021,Z 1188.145,A -85,B 0,C 180,E1 3934.944,E2 3934.944} C_VEL
LIN {X 0,Y 36.945,Z 1190.229,A -85,B 0,C 180,E1 3910.505,E2 3910.505} C_VEL
LIN {X 0,Y 32.125,Z 1190.951,A -85,B 0,C 180,E1 3878.953,E2 3878.953} C_VEL
LIN {X 0,Y 32.083,Z 1191.014,A -85,B 0,C 180,E1 3865.804,E2 3865.804} C_VEL
LIN {X 0,Y 34.841,Z 1190.545,A -85,B 0,C 180,E1 3836.957,E2 3836.957} C_VEL
LIN {X 0,Y 50.367,Z 1188.376,A -85,B 0,C 180,E1 3806.707,E2 3806.707} C_VEL
LIN {X 0,Y 69.796,Z 1185.168,A -85,B 0,C 180,E1 3793.061,E2 3793.061} C_VEL
LIN {X 0,Y 90.405,Z 1180.946,A -85,B 0,C 180,E1 3785.513,E2 3785.513} C_VEL
LIN {X 0,Y 112.724,Z 1175.366,A -85,B 0,C 180,E1 3780.508,E2 3780.508} C_VEL
LIN {X 0,Y 121.649,Z 1172.868,A -85,B 0,C 180,E1 3778.999,E2 3778.999} C_VEL
LIN {X 0,Y 94.596,Z 1179.481,A -85,B 0,C 180,E1 3773.492,E2 3773.492} C_VEL
LIN {X 0,Y 73.103,Z 1183.596,A -85,B 0,C 180,E1 3766.188,E2 3766.188} C_VEL
LIN {X 0,Y 55.073,Z 1186.304,A -85,B 0,C 180,E1 3755.197,E2 3755.197} C_VEL
LIN {X 0,Y 40.904,Z 1187.967,A -85,B 0,C 180,E1 3737.166,E2 3737.166} C_VEL
LIN {X 0,Y 33.337,Z 1188.723,A -85,B 0,C 180,E1 3711.094,E2 3711.094} C_VEL
LIN {X 0,Y 32.128,Z 1188.947,A -85,B 0,C 180,E1 3688.217,E2 3688.217} C_VEL
LIN {X 0,Y 34.101,Z 1188.678,A -85,B 0,C 180,E1 3663.909,E2 3663.909} C_VEL
LIN {X 0,Y 46.026,Z 1187.504,A -85,B 0,C 180,E1 3634.361,E2 3634.361} C_VEL
LIN {X 0,Y 68.606,Z 1184.399,A -85,B 0,C 180,E1 3615.873,E2 3615.873} C_VEL
LIN {X 0,Y 89.805,Z 1180.528,A -85,B 0,C 180,E1 3607.737,E2 3607.737} C_VEL
LIN {X 0,Y 111.111,Z 1175.672,A -85,B 0,C 180,E1 3602.737,E2 3602.737} C_VEL
LIN {X 0,Y 121.481,Z 1173.007,A -85,B 0,C 180,E1 3600.943,E2 3600.943} C_VEL
LIN {X 0,Y 94.274,Z 1180.132,A -85,B 0,C 180,E1 3595.524,E2 3595.524} C_VEL
LIN {X 0,Y 72.522,Z 1184.701,A -85,B 0,C 180,E1 3588.199,E2 3588.199} C_VEL
LIN {X 0,Y 54.305,Z 1187.792,A -85,B 0,C 180,E1 3577.014,E2 3577.014} C_VEL
LIN {X 0,Y 52.021,Z 1188.145,A -85,B 0,C 180,E1 3574.944,E2 3574.944} C_VEL
LIN {X 0,Y 45.771,Z 1189.013,A -85,B 0,C 180,E1 3569.629,E2 3569.629} C_VEL
LIN {X 0,Y 27.539,Z 1190.387,A -85,B 0,C 180,E1 3546.98,E2 3546.98} C_VEL
LIN {X 0,Y 25.338,Z 1190.501,A -85,B 0,C 180,E1 3537.145,E2 3537.145} C_VEL
LIN {X 0,Y 24.118,Z 1190.805,A -85,B 0,C 180,E1 3510,E2 3510} C_VEL
LIN {X 0,Y 25.467,Z 1190.482,A -85,B 0,C 180,E1 3481.893,E2 3481.893} C_VEL
LIN {X 0,Y 35.182,Z 1189.484,A -85,B 0,C 180,E1 3451.506,E2 3451.506} C_VEL
LIN {X 0,Y 51.623,Z 1187.487,A -85,B 0,C 180,E1 3434.437,E2 3434.437} C_VEL
LIN {X 0,Y 71.281,Z 1184.382,A -85,B 0,C 180,E1 3425.183,E2 3425.183} C_VEL
LIN {X 0,Y 93.993,Z 1179.798,A -85,B 0,C 180,E1 3419.338,E2 3419.338} C_VEL
LIN {X 0,Y 96.003,Z 1179.362,A -85,B 0,C 180,E1 3418.935,E2 3418.935} C_VEL
LIN {X 0,Y 72.138,Z 1183.781,A -85,B 0,C 180,E1 3412.834,E2 3412.834} C_VEL
LIN {X 0,Y 52.154,Z 1186.575,A -85,B 0,C 180,E1 3403.448,E2 3403.448} C_VEL
LIN {X 0,Y 35.852,Z 1188.235,A -85,B 0,C 180,E1 3386.788,E2 3386.788} C_VEL
LIN {X 0,Y 25.959,Z 1188.989,A -85,B 0,C 180,E1 3357.529,E2 3357.529} C_VEL
LIN {X 0,Y 24.135,Z 1189.221,A -85,B 0,C 180,E1 3330,E2 3330} C_VEL
LIN {X 0,Y 26.287,Z 1188.979,A -85,B 0,C 180,E1 3300.365,E2 3300.365} C_VEL
LIN {X 0,Y 37.811,Z 1188.093,A -85,B 0,C 180,E1 3270.162,E2 3270.162} C_VEL
LIN {X 0,Y 58.266,Z 1185.897,A -85,B 0,C 180,E1 3252.891,E2 3252.891} C_VEL
LIN {X 0,Y 85.133,Z 1181.588,A -85,B 0,C 180,E1 3243.348,E2 3243.348} C_VEL
LIN {X 0,Y 95.799,Z 1179.464,A -85,B 0,C 180,E1 3241.004,E2 3241.004} C_VEL
LIN {X 0,Y 72.25,Z 1184.256,A -85,B 0,C 180,E1 3235.137,E2 3235.137} C_VEL
LIN {X 0,Y 52.521,Z 1187.395,A -85,B 0,C 180,E1 3226.145,E2 3226.145} C_VEL
LIN {X 0,Y 35.907,Z 1189.426,A -85,B 0,C 180,E1 3209.68,E2 3209.68} C_VEL
LIN {X 0,Y 25.786,Z 1190.459,A -85,B 0,C 180,E1 3180.271,E2 3180.271} C_VEL
LIN {X 0,Y 25.338,Z 1190.501,A -85,B 0,C 180,E1 3177.145,E2 3177.145} C_VEL
LIN {X 0,Y 23.313,Z 1190.654,A -85,B 0,C 180,E1 3163.679,E2 3163.679} C_VEL
LIN {X 0,Y 20.754,Z 1190.66,A -85,B 0,C 180,E1 3144.381,E2 3144.381} C_VEL
LIN {X 0,Y 23.697,Z 1189.974,A -85,B 0,C 180,E1 3092.517,E2 3092.517} C_VEL
LIN {X 0,Y 25.7,Z 1189.765,A -85,B 0,C 180,E1 3087.675,E2 3087.675} C_VEL
LIN {X 0,Y 46.346,Z 1187.706,A -85,B 0,C 180,E1 3067.071,E2 3067.071} C_VEL
LIN {X 0,Y 67.998,Z 1184.616,A -85,B 0,C 180,E1 3059.156,E2 3059.156} C_VEL
LIN {X 0,Y 69.005,Z 1184.442,A -85,B 0,C 180,E1 3058.804,E2 3058.804} C_VEL
LIN {X 0,Y 47.57,Z 1187.162,A -85,B 0,C 180,E1 3051.07,E2 3051.07} C_VEL
LIN {X 0,Y 26.153,Z 1188.95,A -85,B 0,C 180,E1 3030.197,E2 3030.197} C_VEL
LIN {X 0,Y 16.613,Z 1189.383,A -85,B 0,C 180,E1 2987.513,E2 2987.513} C_VEL
LIN {X 0,Y 16.293,Z 1189.428,A -85,B 0,C 180,E1 2959.08,E2 2959.08} C_VEL
LIN {X 0,Y 24.129,Z 1189.124,A -85,B 0,C 180,E1 2914.03,E2 2914.03} C_VEL
LIN {X 0,Y 46.613,Z 1187.303,A -85,B 0,C 180,E1 2889.353,E2 2889.353} C_VEL
LIN {X 0,Y 68.009,Z 1184.641,A -85,B 0,C 180,E1 2881.367,E2 2881.367} C_VEL
LIN {X 0,Y 69.002,Z 1184.492,A -85,B 0,C 180,E1 2881.093,E2 2881.093} C_VEL
LIN {X 0,Y 47.304,Z 1187.615,A -85,B 0,C 180,E1 2873.427,E2 2873.427} C_VEL
LIN {X 0,Y 25.502,Z 1189.803,A -85,B 0,C 180,E1 2851.933,E2 2851.933} C_VEL
LIN {X 0,Y 16.145,Z 1190.476,A -85,B 0,C 180,E1 2800.707,E2 2800.707} C_VEL
LIN {X 0,Y 16.094,Z 1190.496,A -85,B 0,C 180,E1 2782.862,E2 2782.862} C_VEL
LIN {X 0,Y 24.365,Z 1189.899,A -85,B 0,C 180,E1 2730.486,E2 2730.486} C_VEL
LIN {X 0,Y 25.7,Z 1189.765,A -85,B 0,C 180,E1 2727.675,E2 2727.675} C_VEL
LIN {X 0,Y 25.961,Z 1189.651,A -85,B 0,C 180,E1 2723.759,E2 2723.759} C_VEL
LIN {X 0,Y 24.255,Z 1189.583,A -85,B 0,C 180,E1 2717.255,E2 2717.255} C_VEL
LIN {X 0,Y 20.195,Z 1189.644,A -85,B 0,C 180,E1 2707.719,E2 2707.719} C_VEL
LIN {X 0,Y 13.676,Z 1189.701,A -85,B 0,C 180,E1 2690.358,E2 2690.358} C_VEL
LIN {X 0,Y 8.581,Z 1189.762,A -85,B 0,C 180,E1 2651.601,E2 2651.601} C_VEL
LIN {X 0,Y 7.957,Z 1189.749,A -85,B 0,C 180,E1 2605.824,E2 2605.824} C_VEL
LIN {X 0,Y 8.661,Z 1189.684,A -85,B 0,C 180,E1 2586.581,E2 2586.581} C_VEL
LIN {X 0,Y 22.548,Z 1189.282,A -85,B 0,C 180,E1 2532.701,E2 2532.701} C_VEL
LIN {X 0,Y 39.907,Z 1188.197,A -85,B 0,C 180,E1 2521.238,E2 2521.238} C_VEL
LIN {X 0,Y 15.984,Z 1189.864,A -85,B 0,C 180,E1 2499.771,E2 2499.771} C_VEL
LIN {X 0,Y 8.105,Z 1190.279,A -85,B 0,C 180,E1 2430,E2 2430} C_VEL
LIN {X 0,Y 16.854,Z 1189.828,A -85,B 0,C 180,E1 2358.346,E2 2358.346} C_VEL
LIN {X 0,Y 40.005,Z 1188.164,A -85,B 0,C 180,E1 2338.701,E2 2338.701} C_VEL
LIN {X 0,Y 16.273,Z 1189.469,A -85,B 0,C 180,E1 2317.164,E2 2317.164} C_VEL
LIN {X 0,Y 8.17,Z 1189.728,A -85,B 0,C 180,E1 2257.03,E2 2257.03} C_VEL
LIN {X 0,Y 8.661,Z 1189.684,A -85,B 0,C 180,E1 2226.581,E2 2226.581} C_VEL
LIN {X 0,Y 7.641,Z 1189.726,A -85,B 0,C 180,E1 2222.787,E2 2222.787} C_VEL
LIN {X 0,Y 1.828,Z 1189.95,A -85,B 0,C 180,E1 2306.251,E2 2306.251} C_VEL
LIN {X 0,Y 1.354,Z 1189.984,A -85,B 0,C 180,E1 2337.711,E2 2337.711} C_VEL
LIN {X 0,Y 1.343,Z 1189.991,A -85,B 0,C 180,E1 2162.277,E2 2162.277} C_VEL
LIN {X 0,Y 1.354,Z 1189.984,A -85,B 0,C 180,E1 2337.711,E2 2337.711} C_VEL
LIN {X 0,Y 3.377,Z 1191.984,A -85,B 0,C 180,E1 2343.779,E2 2343.779} C_VEL
LIN {X 0,Y 3.377,Z 1215,A -85,B 0,C 180,E1 2343.779,E2 2343.779} C_VEL
LIN {X 0,Y 3.377,Z 1215,A -85,B 0,C 180,E1 2343.779,E2 2343.779}

QRS_NEXT_CUT()

QRS_NEXT()
QRS_HOME()

END
